// TIA Portal V17 export
// export: Created 2025-06-20T10:18:23.2551745Z, ExportSetting WithDefaults, DisplayName Totally Integrated Automation Portal, DisplayVersion V17 Update 8, DisplayName TIA Portal Openness, DisplayVersion V17 Update 8, DisplayName TIA Portal Version Control Interface, DisplayVersion V17, DisplayName SINAMICS Startdrive Advanced, DisplayVersion V17 SP2, DisplayName SINAMICS Startdrive G110M, G120, G120C, G120D, G120P, G115D, DisplayVersion V17 SP2, DisplayName SINAMICS Startdrive G130, G150, S120, S150, SINAMICS MV, S210, DisplayVersion V17 SP2, DisplayName STEP 7 Professional, DisplayVersion V17 Update 8, DisplayName SINUMERIK ONE STEP 7 Toolbox, DisplayVersion V17 Update 12, DisplayName SINUMERIK ONE PLC Basic Program Plus, DisplayVersion V17 Update 12, DisplayName SINUMERIK 840D sl STEP 7 Toolbox, DisplayVersion V17 Update 12, DisplayName STEP 7 Safety, DisplayVersion V17 Update 6, DisplayName WinCC Advanced, DisplayVersion V17 Update 8
FUNCTION "FC17000_MAIN_MAINTENANCE" : Void   // FC17000, LAD
{ S7_Optimized_Access := 'TRUE' }
VERSION : 0.1
// stored: AutoNumber false, IsIECCheckEnabled false, SetENOAutomatically false, UDAEnableTagReadback false
   VAR_TEMP
      ONLY_ONE_MAINT : Bool;
      NULL : Bool;
   END_VAR
BEGIN

REGION Network 1: CALL FC17100 MAINTENANCE HMI SCREEN VARIABLES
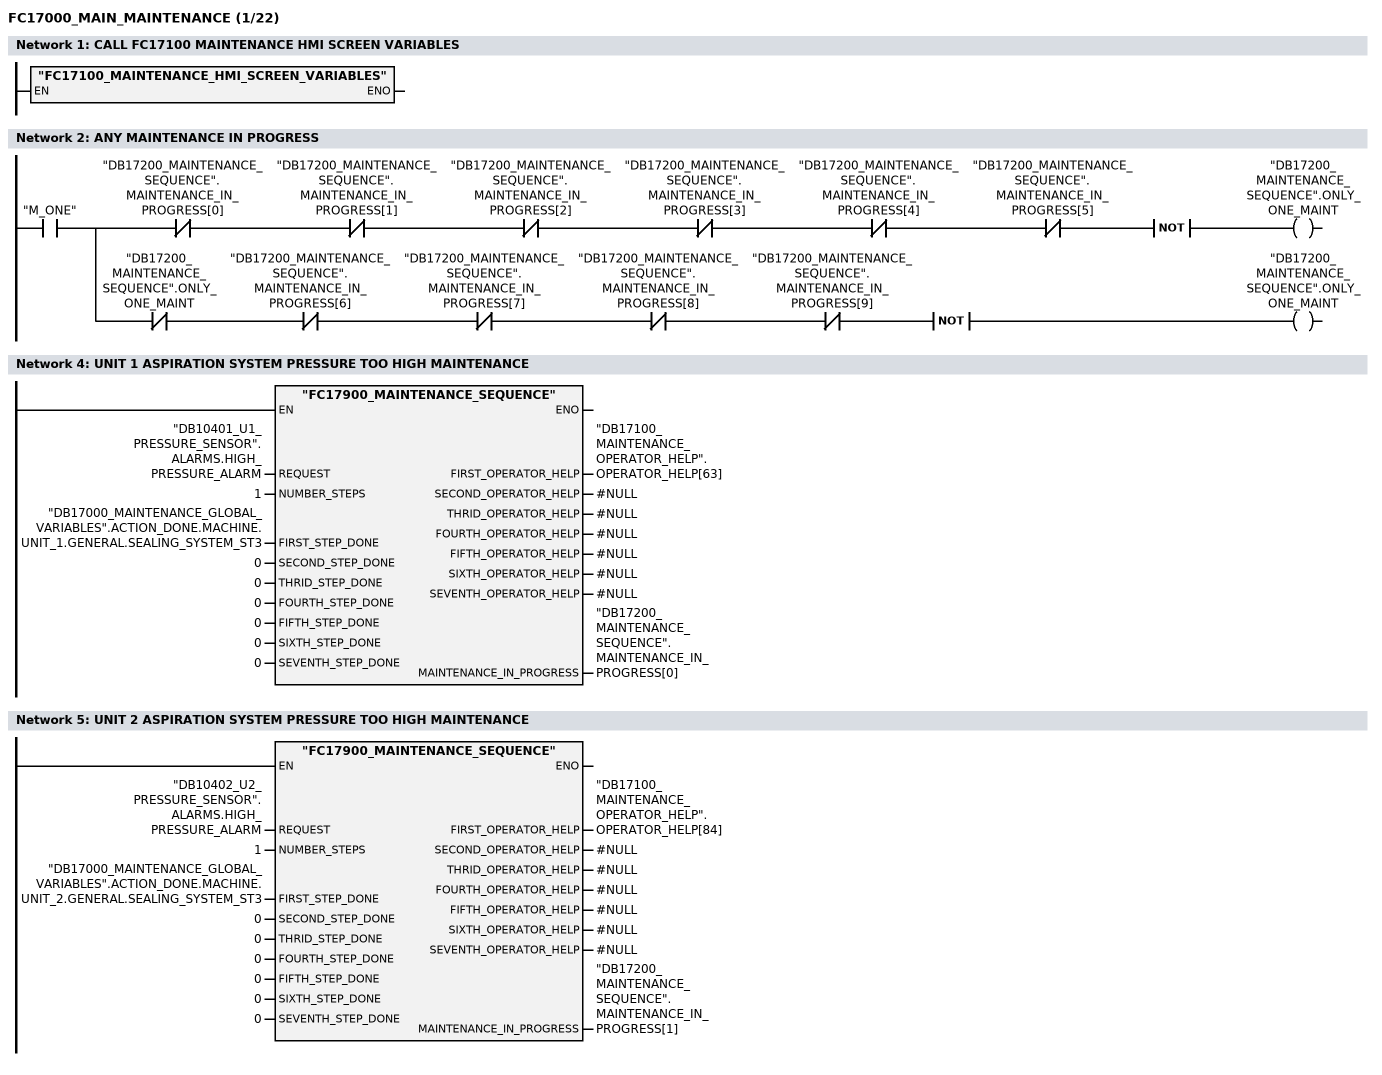
   RUNG wire#powerrail
      "FC17100_MAINTENANCE_HMI_SCREEN_VARIABLES"()
   END_RUNG
   // the same network as SCL:
   "FC17100_MAINTENANCE_HMI_SCREEN_VARIABLES"();
END_REGION

REGION Network 2: ANY MAINTENANCE IN PROGRESS
   RUNG wire#powerrail
      Contact( "M_ONE" )
      wire#w1
      I_Contact( "DB17200_MAINTENANCE_SEQUENCE".MAINTENANCE_IN_PROGRESS[0] )
      I_Contact( "DB17200_MAINTENANCE_SEQUENCE".MAINTENANCE_IN_PROGRESS[1] )
      I_Contact( "DB17200_MAINTENANCE_SEQUENCE".MAINTENANCE_IN_PROGRESS[2] )
      I_Contact( "DB17200_MAINTENANCE_SEQUENCE".MAINTENANCE_IN_PROGRESS[3] )
      I_Contact( "DB17200_MAINTENANCE_SEQUENCE".MAINTENANCE_IN_PROGRESS[4] )
      I_Contact( "DB17200_MAINTENANCE_SEQUENCE".MAINTENANCE_IN_PROGRESS[5] )
      Not()
      Coil( "DB17200_MAINTENANCE_SEQUENCE".ONLY_ONE_MAINT )
   END_RUNG
   RUNG wire#w1
      I_Contact( "DB17200_MAINTENANCE_SEQUENCE".ONLY_ONE_MAINT )
      I_Contact( "DB17200_MAINTENANCE_SEQUENCE".MAINTENANCE_IN_PROGRESS[6] )
      I_Contact( "DB17200_MAINTENANCE_SEQUENCE".MAINTENANCE_IN_PROGRESS[7] )
      I_Contact( "DB17200_MAINTENANCE_SEQUENCE".MAINTENANCE_IN_PROGRESS[8] )
      I_Contact( "DB17200_MAINTENANCE_SEQUENCE".MAINTENANCE_IN_PROGRESS[9] )
      Not()
      Coil( "DB17200_MAINTENANCE_SEQUENCE".ONLY_ONE_MAINT )
   END_RUNG
   // the same network as SCL:
   "DB17200_MAINTENANCE_SEQUENCE".ONLY_ONE_MAINT := NOT ("M_ONE" AND NOT "DB17200_MAINTENANCE_SEQUENCE".MAINTENANCE_IN_PROGRESS[0] AND NOT "DB17200_MAINTENANCE_SEQUENCE".MAINTENANCE_IN_PROGRESS[1] AND NOT "DB17200_MAINTENANCE_SEQUENCE".MAINTENANCE_IN_PROGRESS[2] AND NOT "DB17200_MAINTENANCE_SEQUENCE".MAINTENANCE_IN_PROGRESS[3] AND NOT "DB17200_MAINTENANCE_SEQUENCE".MAINTENANCE_IN_PROGRESS[4] AND NOT "DB17200_MAINTENANCE_SEQUENCE".MAINTENANCE_IN_PROGRESS[5]);
   "DB17200_MAINTENANCE_SEQUENCE".ONLY_ONE_MAINT := NOT ("M_ONE" AND NOT "DB17200_MAINTENANCE_SEQUENCE".ONLY_ONE_MAINT AND NOT "DB17200_MAINTENANCE_SEQUENCE".MAINTENANCE_IN_PROGRESS[6] AND NOT "DB17200_MAINTENANCE_SEQUENCE".MAINTENANCE_IN_PROGRESS[7] AND NOT "DB17200_MAINTENANCE_SEQUENCE".MAINTENANCE_IN_PROGRESS[8] AND NOT "DB17200_MAINTENANCE_SEQUENCE".MAINTENANCE_IN_PROGRESS[9]);
END_REGION

REGION Network 3: <<<---ALARMS--->>>
END_REGION

REGION Network 4: UNIT 1 ASPIRATION SYSTEM PRESSURE TOO HIGH MAINTENANCE
   RUNG wire#powerrail
      "FC17900_MAINTENANCE_SEQUENCE"(REQUEST := "DB10401_U1_PRESSURE_SENSOR".ALARMS.HIGH_PRESSURE_ALARM, NUMBER_STEPS := 1, FIRST_STEP_DONE := "DB17000_MAINTENANCE_GLOBAL_VARIABLES".ACTION_DONE.MACHINE.UNIT_1.GENERAL.SEALING_SYSTEM_ST3, SECOND_STEP_DONE := 0, THRID_STEP_DONE := 0, FOURTH_STEP_DONE := 0, FIFTH_STEP_DONE := 0, SIXTH_STEP_DONE := 0, SEVENTH_STEP_DONE := 0, FIRST_OPERATOR_HELP => "DB17100_MAINTENANCE_OPERATOR_HELP".OPERATOR_HELP[63], SECOND_OPERATOR_HELP => #NULL, THRID_OPERATOR_HELP => #NULL, FOURTH_OPERATOR_HELP => #NULL, FIFTH_OPERATOR_HELP => #NULL, SIXTH_OPERATOR_HELP => #NULL, SEVENTH_OPERATOR_HELP => #NULL, MAINTENANCE_IN_PROGRESS => "DB17200_MAINTENANCE_SEQUENCE".MAINTENANCE_IN_PROGRESS[0])
   END_RUNG
   // the same network as SCL:
   "FC17900_MAINTENANCE_SEQUENCE"(REQUEST := "DB10401_U1_PRESSURE_SENSOR".ALARMS.HIGH_PRESSURE_ALARM,
                           NUMBER_STEPS := 1,
                           FIRST_STEP_DONE := "DB17000_MAINTENANCE_GLOBAL_VARIABLES".ACTION_DONE.MACHINE.UNIT_1.GENERAL.SEALING_SYSTEM_ST3,
                           SECOND_STEP_DONE := 0,
                           THRID_STEP_DONE := 0,
                           FOURTH_STEP_DONE := 0,
                           FIFTH_STEP_DONE := 0,
                           SIXTH_STEP_DONE := 0,
                           SEVENTH_STEP_DONE := 0,
                           FIRST_OPERATOR_HELP => "DB17100_MAINTENANCE_OPERATOR_HELP".OPERATOR_HELP[63],
                           SECOND_OPERATOR_HELP => #NULL,
                           THRID_OPERATOR_HELP => #NULL,
                           FOURTH_OPERATOR_HELP => #NULL,
                           FIFTH_OPERATOR_HELP => #NULL,
                           SIXTH_OPERATOR_HELP => #NULL,
                           SEVENTH_OPERATOR_HELP => #NULL,
                           MAINTENANCE_IN_PROGRESS => "DB17200_MAINTENANCE_SEQUENCE".MAINTENANCE_IN_PROGRESS[0]);
END_REGION

REGION Network 5: UNIT 2 ASPIRATION SYSTEM PRESSURE TOO HIGH MAINTENANCE
   RUNG wire#powerrail
      "FC17900_MAINTENANCE_SEQUENCE"(REQUEST := "DB10402_U2_PRESSURE_SENSOR".ALARMS.HIGH_PRESSURE_ALARM, NUMBER_STEPS := 1, FIRST_STEP_DONE := "DB17000_MAINTENANCE_GLOBAL_VARIABLES".ACTION_DONE.MACHINE.UNIT_2.GENERAL.SEALING_SYSTEM_ST3, SECOND_STEP_DONE := 0, THRID_STEP_DONE := 0, FOURTH_STEP_DONE := 0, FIFTH_STEP_DONE := 0, SIXTH_STEP_DONE := 0, SEVENTH_STEP_DONE := 0, FIRST_OPERATOR_HELP => "DB17100_MAINTENANCE_OPERATOR_HELP".OPERATOR_HELP[84], SECOND_OPERATOR_HELP => #NULL, THRID_OPERATOR_HELP => #NULL, FOURTH_OPERATOR_HELP => #NULL, FIFTH_OPERATOR_HELP => #NULL, SIXTH_OPERATOR_HELP => #NULL, SEVENTH_OPERATOR_HELP => #NULL, MAINTENANCE_IN_PROGRESS => "DB17200_MAINTENANCE_SEQUENCE".MAINTENANCE_IN_PROGRESS[1])
   END_RUNG
   // the same network as SCL:
   "FC17900_MAINTENANCE_SEQUENCE"(REQUEST := "DB10402_U2_PRESSURE_SENSOR".ALARMS.HIGH_PRESSURE_ALARM,
                           NUMBER_STEPS := 1,
                           FIRST_STEP_DONE := "DB17000_MAINTENANCE_GLOBAL_VARIABLES".ACTION_DONE.MACHINE.UNIT_2.GENERAL.SEALING_SYSTEM_ST3,
                           SECOND_STEP_DONE := 0,
                           THRID_STEP_DONE := 0,
                           FOURTH_STEP_DONE := 0,
                           FIFTH_STEP_DONE := 0,
                           SIXTH_STEP_DONE := 0,
                           SEVENTH_STEP_DONE := 0,
                           FIRST_OPERATOR_HELP => "DB17100_MAINTENANCE_OPERATOR_HELP".OPERATOR_HELP[84],
                           SECOND_OPERATOR_HELP => #NULL,
                           THRID_OPERATOR_HELP => #NULL,
                           FOURTH_OPERATOR_HELP => #NULL,
                           FIFTH_OPERATOR_HELP => #NULL,
                           SIXTH_OPERATOR_HELP => #NULL,
                           SEVENTH_OPERATOR_HELP => #NULL,
                           MAINTENANCE_IN_PROGRESS => "DB17200_MAINTENANCE_SEQUENCE".MAINTENANCE_IN_PROGRESS[1]);
END_REGION

REGION Network 6: UNIT 1 FIXTURE 1 NOT CLAMPED
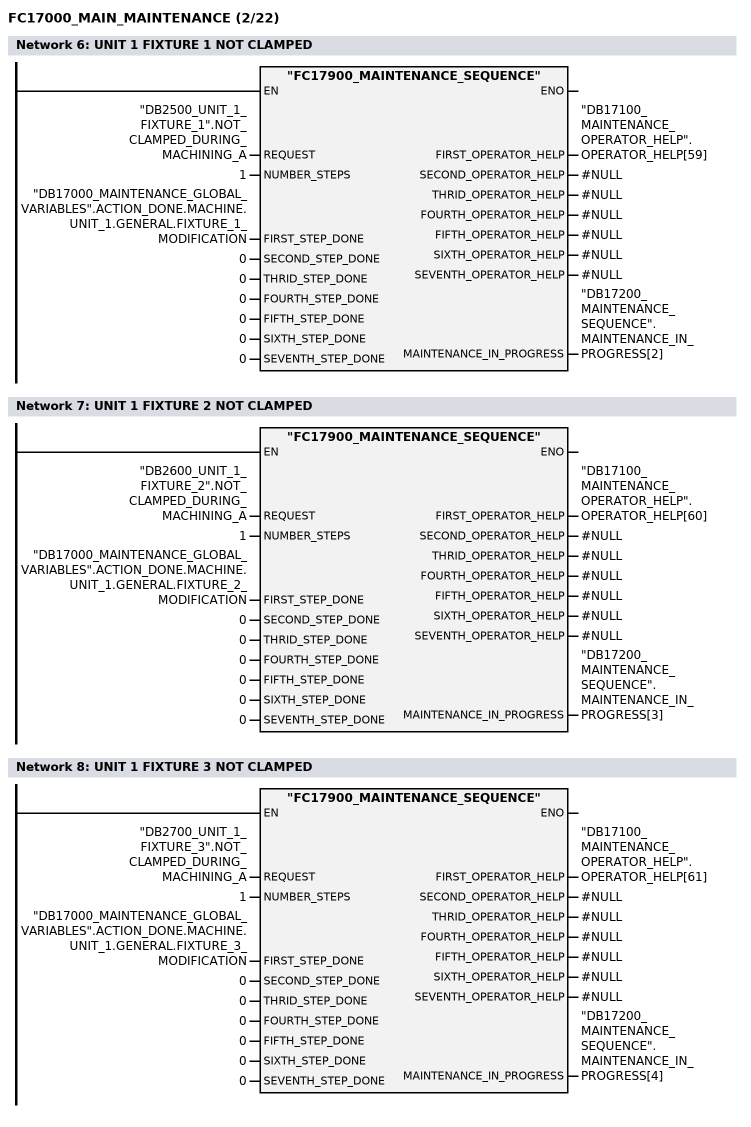
   RUNG wire#powerrail
      "FC17900_MAINTENANCE_SEQUENCE"(REQUEST := "DB2500_UNIT_1_FIXTURE_1".NOT_CLAMPED_DURING_MACHINING_A, NUMBER_STEPS := 1, FIRST_STEP_DONE := "DB17000_MAINTENANCE_GLOBAL_VARIABLES".ACTION_DONE.MACHINE.UNIT_1.GENERAL.FIXTURE_1_MODIFICATION, SECOND_STEP_DONE := 0, THRID_STEP_DONE := 0, FOURTH_STEP_DONE := 0, FIFTH_STEP_DONE := 0, SIXTH_STEP_DONE := 0, SEVENTH_STEP_DONE := 0, FIRST_OPERATOR_HELP => "DB17100_MAINTENANCE_OPERATOR_HELP".OPERATOR_HELP[59], SECOND_OPERATOR_HELP => #NULL, THRID_OPERATOR_HELP => #NULL, FOURTH_OPERATOR_HELP => #NULL, FIFTH_OPERATOR_HELP => #NULL, SIXTH_OPERATOR_HELP => #NULL, SEVENTH_OPERATOR_HELP => #NULL, MAINTENANCE_IN_PROGRESS => "DB17200_MAINTENANCE_SEQUENCE".MAINTENANCE_IN_PROGRESS[2])
   END_RUNG
   // the same network as SCL:
   "FC17900_MAINTENANCE_SEQUENCE"(REQUEST := "DB2500_UNIT_1_FIXTURE_1".NOT_CLAMPED_DURING_MACHINING_A,
                           NUMBER_STEPS := 1,
                           FIRST_STEP_DONE := "DB17000_MAINTENANCE_GLOBAL_VARIABLES".ACTION_DONE.MACHINE.UNIT_1.GENERAL.FIXTURE_1_MODIFICATION,
                           SECOND_STEP_DONE := 0,
                           THRID_STEP_DONE := 0,
                           FOURTH_STEP_DONE := 0,
                           FIFTH_STEP_DONE := 0,
                           SIXTH_STEP_DONE := 0,
                           SEVENTH_STEP_DONE := 0,
                           FIRST_OPERATOR_HELP => "DB17100_MAINTENANCE_OPERATOR_HELP".OPERATOR_HELP[59],
                           SECOND_OPERATOR_HELP => #NULL,
                           THRID_OPERATOR_HELP => #NULL,
                           FOURTH_OPERATOR_HELP => #NULL,
                           FIFTH_OPERATOR_HELP => #NULL,
                           SIXTH_OPERATOR_HELP => #NULL,
                           SEVENTH_OPERATOR_HELP => #NULL,
                           MAINTENANCE_IN_PROGRESS => "DB17200_MAINTENANCE_SEQUENCE".MAINTENANCE_IN_PROGRESS[2]);
END_REGION

REGION Network 7: UNIT 1 FIXTURE 2 NOT CLAMPED
   RUNG wire#powerrail
      "FC17900_MAINTENANCE_SEQUENCE"(REQUEST := "DB2600_UNIT_1_FIXTURE_2".NOT_CLAMPED_DURING_MACHINING_A, NUMBER_STEPS := 1, FIRST_STEP_DONE := "DB17000_MAINTENANCE_GLOBAL_VARIABLES".ACTION_DONE.MACHINE.UNIT_1.GENERAL.FIXTURE_2_MODIFICATION, SECOND_STEP_DONE := 0, THRID_STEP_DONE := 0, FOURTH_STEP_DONE := 0, FIFTH_STEP_DONE := 0, SIXTH_STEP_DONE := 0, SEVENTH_STEP_DONE := 0, FIRST_OPERATOR_HELP => "DB17100_MAINTENANCE_OPERATOR_HELP".OPERATOR_HELP[60], SECOND_OPERATOR_HELP => #NULL, THRID_OPERATOR_HELP => #NULL, FOURTH_OPERATOR_HELP => #NULL, FIFTH_OPERATOR_HELP => #NULL, SIXTH_OPERATOR_HELP => #NULL, SEVENTH_OPERATOR_HELP => #NULL, MAINTENANCE_IN_PROGRESS => "DB17200_MAINTENANCE_SEQUENCE".MAINTENANCE_IN_PROGRESS[3])
   END_RUNG
   // the same network as SCL:
   "FC17900_MAINTENANCE_SEQUENCE"(REQUEST := "DB2600_UNIT_1_FIXTURE_2".NOT_CLAMPED_DURING_MACHINING_A,
                           NUMBER_STEPS := 1,
                           FIRST_STEP_DONE := "DB17000_MAINTENANCE_GLOBAL_VARIABLES".ACTION_DONE.MACHINE.UNIT_1.GENERAL.FIXTURE_2_MODIFICATION,
                           SECOND_STEP_DONE := 0,
                           THRID_STEP_DONE := 0,
                           FOURTH_STEP_DONE := 0,
                           FIFTH_STEP_DONE := 0,
                           SIXTH_STEP_DONE := 0,
                           SEVENTH_STEP_DONE := 0,
                           FIRST_OPERATOR_HELP => "DB17100_MAINTENANCE_OPERATOR_HELP".OPERATOR_HELP[60],
                           SECOND_OPERATOR_HELP => #NULL,
                           THRID_OPERATOR_HELP => #NULL,
                           FOURTH_OPERATOR_HELP => #NULL,
                           FIFTH_OPERATOR_HELP => #NULL,
                           SIXTH_OPERATOR_HELP => #NULL,
                           SEVENTH_OPERATOR_HELP => #NULL,
                           MAINTENANCE_IN_PROGRESS => "DB17200_MAINTENANCE_SEQUENCE".MAINTENANCE_IN_PROGRESS[3]);
END_REGION

REGION Network 8: UNIT 1 FIXTURE 3 NOT CLAMPED
   RUNG wire#powerrail
      "FC17900_MAINTENANCE_SEQUENCE"(REQUEST := "DB2700_UNIT_1_FIXTURE_3".NOT_CLAMPED_DURING_MACHINING_A, NUMBER_STEPS := 1, FIRST_STEP_DONE := "DB17000_MAINTENANCE_GLOBAL_VARIABLES".ACTION_DONE.MACHINE.UNIT_1.GENERAL.FIXTURE_3_MODIFICATION, SECOND_STEP_DONE := 0, THRID_STEP_DONE := 0, FOURTH_STEP_DONE := 0, FIFTH_STEP_DONE := 0, SIXTH_STEP_DONE := 0, SEVENTH_STEP_DONE := 0, FIRST_OPERATOR_HELP => "DB17100_MAINTENANCE_OPERATOR_HELP".OPERATOR_HELP[61], SECOND_OPERATOR_HELP => #NULL, THRID_OPERATOR_HELP => #NULL, FOURTH_OPERATOR_HELP => #NULL, FIFTH_OPERATOR_HELP => #NULL, SIXTH_OPERATOR_HELP => #NULL, SEVENTH_OPERATOR_HELP => #NULL, MAINTENANCE_IN_PROGRESS => "DB17200_MAINTENANCE_SEQUENCE".MAINTENANCE_IN_PROGRESS[4])
   END_RUNG
   // the same network as SCL:
   "FC17900_MAINTENANCE_SEQUENCE"(REQUEST := "DB2700_UNIT_1_FIXTURE_3".NOT_CLAMPED_DURING_MACHINING_A,
                           NUMBER_STEPS := 1,
                           FIRST_STEP_DONE := "DB17000_MAINTENANCE_GLOBAL_VARIABLES".ACTION_DONE.MACHINE.UNIT_1.GENERAL.FIXTURE_3_MODIFICATION,
                           SECOND_STEP_DONE := 0,
                           THRID_STEP_DONE := 0,
                           FOURTH_STEP_DONE := 0,
                           FIFTH_STEP_DONE := 0,
                           SIXTH_STEP_DONE := 0,
                           SEVENTH_STEP_DONE := 0,
                           FIRST_OPERATOR_HELP => "DB17100_MAINTENANCE_OPERATOR_HELP".OPERATOR_HELP[61],
                           SECOND_OPERATOR_HELP => #NULL,
                           THRID_OPERATOR_HELP => #NULL,
                           FOURTH_OPERATOR_HELP => #NULL,
                           FIFTH_OPERATOR_HELP => #NULL,
                           SIXTH_OPERATOR_HELP => #NULL,
                           SEVENTH_OPERATOR_HELP => #NULL,
                           MAINTENANCE_IN_PROGRESS => "DB17200_MAINTENANCE_SEQUENCE".MAINTENANCE_IN_PROGRESS[4]);
END_REGION

REGION Network 9: UNIT 1 FIXTURE 4 NOT CLAMPED
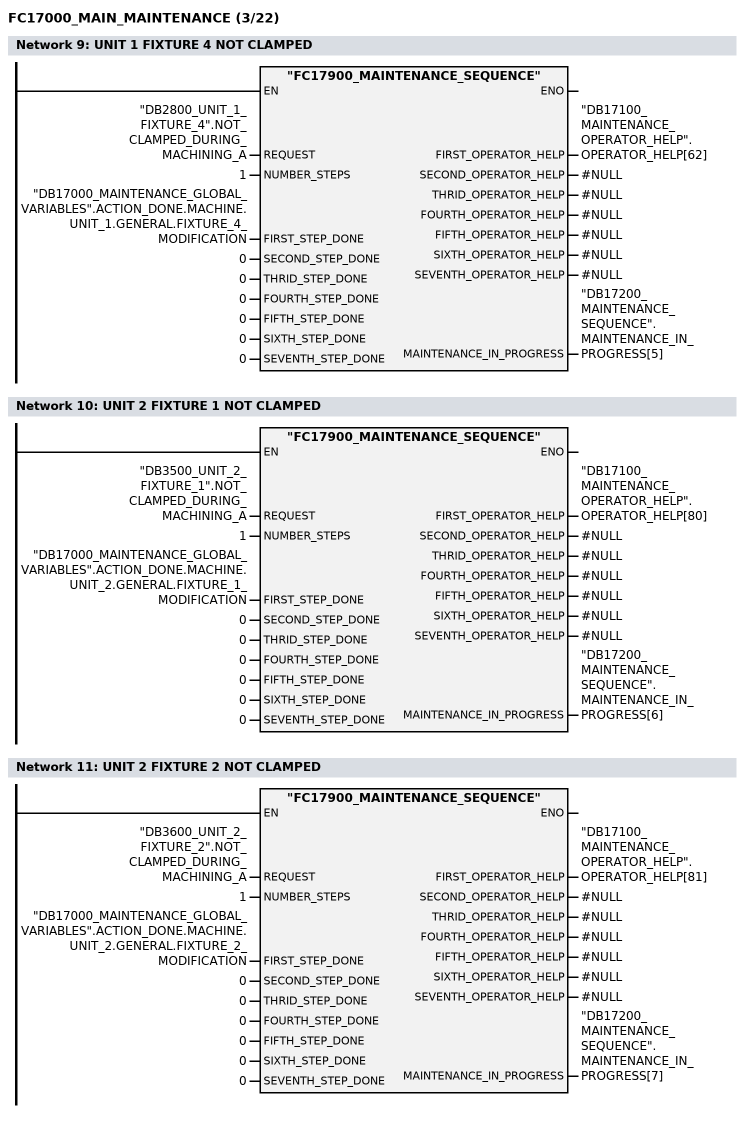
   RUNG wire#powerrail
      "FC17900_MAINTENANCE_SEQUENCE"(REQUEST := "DB2800_UNIT_1_FIXTURE_4".NOT_CLAMPED_DURING_MACHINING_A, NUMBER_STEPS := 1, FIRST_STEP_DONE := "DB17000_MAINTENANCE_GLOBAL_VARIABLES".ACTION_DONE.MACHINE.UNIT_1.GENERAL.FIXTURE_4_MODIFICATION, SECOND_STEP_DONE := 0, THRID_STEP_DONE := 0, FOURTH_STEP_DONE := 0, FIFTH_STEP_DONE := 0, SIXTH_STEP_DONE := 0, SEVENTH_STEP_DONE := 0, FIRST_OPERATOR_HELP => "DB17100_MAINTENANCE_OPERATOR_HELP".OPERATOR_HELP[62], SECOND_OPERATOR_HELP => #NULL, THRID_OPERATOR_HELP => #NULL, FOURTH_OPERATOR_HELP => #NULL, FIFTH_OPERATOR_HELP => #NULL, SIXTH_OPERATOR_HELP => #NULL, SEVENTH_OPERATOR_HELP => #NULL, MAINTENANCE_IN_PROGRESS => "DB17200_MAINTENANCE_SEQUENCE".MAINTENANCE_IN_PROGRESS[5])
   END_RUNG
   // the same network as SCL:
   "FC17900_MAINTENANCE_SEQUENCE"(REQUEST := "DB2800_UNIT_1_FIXTURE_4".NOT_CLAMPED_DURING_MACHINING_A,
                           NUMBER_STEPS := 1,
                           FIRST_STEP_DONE := "DB17000_MAINTENANCE_GLOBAL_VARIABLES".ACTION_DONE.MACHINE.UNIT_1.GENERAL.FIXTURE_4_MODIFICATION,
                           SECOND_STEP_DONE := 0,
                           THRID_STEP_DONE := 0,
                           FOURTH_STEP_DONE := 0,
                           FIFTH_STEP_DONE := 0,
                           SIXTH_STEP_DONE := 0,
                           SEVENTH_STEP_DONE := 0,
                           FIRST_OPERATOR_HELP => "DB17100_MAINTENANCE_OPERATOR_HELP".OPERATOR_HELP[62],
                           SECOND_OPERATOR_HELP => #NULL,
                           THRID_OPERATOR_HELP => #NULL,
                           FOURTH_OPERATOR_HELP => #NULL,
                           FIFTH_OPERATOR_HELP => #NULL,
                           SIXTH_OPERATOR_HELP => #NULL,
                           SEVENTH_OPERATOR_HELP => #NULL,
                           MAINTENANCE_IN_PROGRESS => "DB17200_MAINTENANCE_SEQUENCE".MAINTENANCE_IN_PROGRESS[5]);
END_REGION

REGION Network 10: UNIT 2 FIXTURE 1 NOT CLAMPED
   RUNG wire#powerrail
      "FC17900_MAINTENANCE_SEQUENCE"(REQUEST := "DB3500_UNIT_2_FIXTURE_1".NOT_CLAMPED_DURING_MACHINING_A, NUMBER_STEPS := 1, FIRST_STEP_DONE := "DB17000_MAINTENANCE_GLOBAL_VARIABLES".ACTION_DONE.MACHINE.UNIT_2.GENERAL.FIXTURE_1_MODIFICATION, SECOND_STEP_DONE := 0, THRID_STEP_DONE := 0, FOURTH_STEP_DONE := 0, FIFTH_STEP_DONE := 0, SIXTH_STEP_DONE := 0, SEVENTH_STEP_DONE := 0, FIRST_OPERATOR_HELP => "DB17100_MAINTENANCE_OPERATOR_HELP".OPERATOR_HELP[80], SECOND_OPERATOR_HELP => #NULL, THRID_OPERATOR_HELP => #NULL, FOURTH_OPERATOR_HELP => #NULL, FIFTH_OPERATOR_HELP => #NULL, SIXTH_OPERATOR_HELP => #NULL, SEVENTH_OPERATOR_HELP => #NULL, MAINTENANCE_IN_PROGRESS => "DB17200_MAINTENANCE_SEQUENCE".MAINTENANCE_IN_PROGRESS[6])
   END_RUNG
   // the same network as SCL:
   "FC17900_MAINTENANCE_SEQUENCE"(REQUEST := "DB3500_UNIT_2_FIXTURE_1".NOT_CLAMPED_DURING_MACHINING_A,
                           NUMBER_STEPS := 1,
                           FIRST_STEP_DONE := "DB17000_MAINTENANCE_GLOBAL_VARIABLES".ACTION_DONE.MACHINE.UNIT_2.GENERAL.FIXTURE_1_MODIFICATION,
                           SECOND_STEP_DONE := 0,
                           THRID_STEP_DONE := 0,
                           FOURTH_STEP_DONE := 0,
                           FIFTH_STEP_DONE := 0,
                           SIXTH_STEP_DONE := 0,
                           SEVENTH_STEP_DONE := 0,
                           FIRST_OPERATOR_HELP => "DB17100_MAINTENANCE_OPERATOR_HELP".OPERATOR_HELP[80],
                           SECOND_OPERATOR_HELP => #NULL,
                           THRID_OPERATOR_HELP => #NULL,
                           FOURTH_OPERATOR_HELP => #NULL,
                           FIFTH_OPERATOR_HELP => #NULL,
                           SIXTH_OPERATOR_HELP => #NULL,
                           SEVENTH_OPERATOR_HELP => #NULL,
                           MAINTENANCE_IN_PROGRESS => "DB17200_MAINTENANCE_SEQUENCE".MAINTENANCE_IN_PROGRESS[6]);
END_REGION

REGION Network 11: UNIT 2 FIXTURE 2 NOT CLAMPED
   RUNG wire#powerrail
      "FC17900_MAINTENANCE_SEQUENCE"(REQUEST := "DB3600_UNIT_2_FIXTURE_2".NOT_CLAMPED_DURING_MACHINING_A, NUMBER_STEPS := 1, FIRST_STEP_DONE := "DB17000_MAINTENANCE_GLOBAL_VARIABLES".ACTION_DONE.MACHINE.UNIT_2.GENERAL.FIXTURE_2_MODIFICATION, SECOND_STEP_DONE := 0, THRID_STEP_DONE := 0, FOURTH_STEP_DONE := 0, FIFTH_STEP_DONE := 0, SIXTH_STEP_DONE := 0, SEVENTH_STEP_DONE := 0, FIRST_OPERATOR_HELP => "DB17100_MAINTENANCE_OPERATOR_HELP".OPERATOR_HELP[81], SECOND_OPERATOR_HELP => #NULL, THRID_OPERATOR_HELP => #NULL, FOURTH_OPERATOR_HELP => #NULL, FIFTH_OPERATOR_HELP => #NULL, SIXTH_OPERATOR_HELP => #NULL, SEVENTH_OPERATOR_HELP => #NULL, MAINTENANCE_IN_PROGRESS => "DB17200_MAINTENANCE_SEQUENCE".MAINTENANCE_IN_PROGRESS[7])
   END_RUNG
   // the same network as SCL:
   "FC17900_MAINTENANCE_SEQUENCE"(REQUEST := "DB3600_UNIT_2_FIXTURE_2".NOT_CLAMPED_DURING_MACHINING_A,
                           NUMBER_STEPS := 1,
                           FIRST_STEP_DONE := "DB17000_MAINTENANCE_GLOBAL_VARIABLES".ACTION_DONE.MACHINE.UNIT_2.GENERAL.FIXTURE_2_MODIFICATION,
                           SECOND_STEP_DONE := 0,
                           THRID_STEP_DONE := 0,
                           FOURTH_STEP_DONE := 0,
                           FIFTH_STEP_DONE := 0,
                           SIXTH_STEP_DONE := 0,
                           SEVENTH_STEP_DONE := 0,
                           FIRST_OPERATOR_HELP => "DB17100_MAINTENANCE_OPERATOR_HELP".OPERATOR_HELP[81],
                           SECOND_OPERATOR_HELP => #NULL,
                           THRID_OPERATOR_HELP => #NULL,
                           FOURTH_OPERATOR_HELP => #NULL,
                           FIFTH_OPERATOR_HELP => #NULL,
                           SIXTH_OPERATOR_HELP => #NULL,
                           SEVENTH_OPERATOR_HELP => #NULL,
                           MAINTENANCE_IN_PROGRESS => "DB17200_MAINTENANCE_SEQUENCE".MAINTENANCE_IN_PROGRESS[7]);
END_REGION

REGION Network 12: UNIT 2 FIXTURE 3 NOT CLAMPED
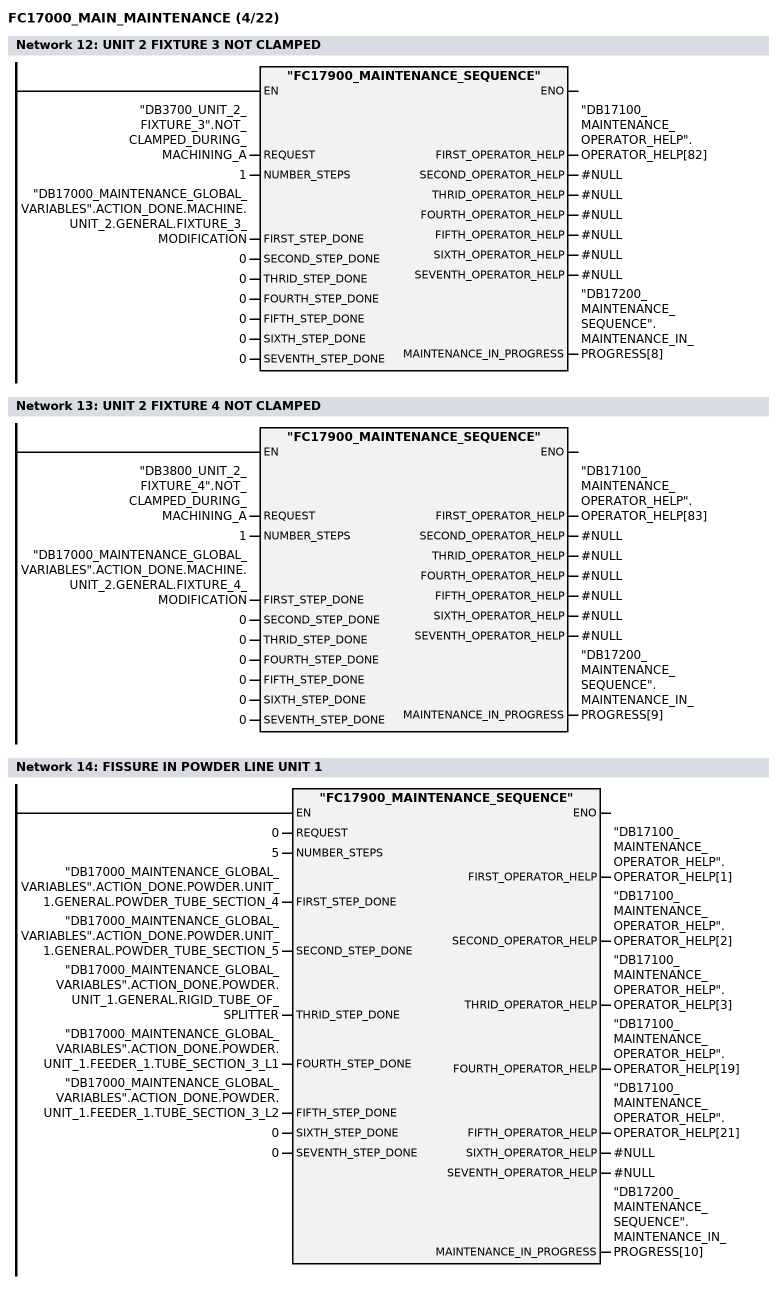
   RUNG wire#powerrail
      "FC17900_MAINTENANCE_SEQUENCE"(REQUEST := "DB3700_UNIT_2_FIXTURE_3".NOT_CLAMPED_DURING_MACHINING_A, NUMBER_STEPS := 1, FIRST_STEP_DONE := "DB17000_MAINTENANCE_GLOBAL_VARIABLES".ACTION_DONE.MACHINE.UNIT_2.GENERAL.FIXTURE_3_MODIFICATION, SECOND_STEP_DONE := 0, THRID_STEP_DONE := 0, FOURTH_STEP_DONE := 0, FIFTH_STEP_DONE := 0, SIXTH_STEP_DONE := 0, SEVENTH_STEP_DONE := 0, FIRST_OPERATOR_HELP => "DB17100_MAINTENANCE_OPERATOR_HELP".OPERATOR_HELP[82], SECOND_OPERATOR_HELP => #NULL, THRID_OPERATOR_HELP => #NULL, FOURTH_OPERATOR_HELP => #NULL, FIFTH_OPERATOR_HELP => #NULL, SIXTH_OPERATOR_HELP => #NULL, SEVENTH_OPERATOR_HELP => #NULL, MAINTENANCE_IN_PROGRESS => "DB17200_MAINTENANCE_SEQUENCE".MAINTENANCE_IN_PROGRESS[8])
   END_RUNG
   // the same network as SCL:
   "FC17900_MAINTENANCE_SEQUENCE"(REQUEST := "DB3700_UNIT_2_FIXTURE_3".NOT_CLAMPED_DURING_MACHINING_A,
                           NUMBER_STEPS := 1,
                           FIRST_STEP_DONE := "DB17000_MAINTENANCE_GLOBAL_VARIABLES".ACTION_DONE.MACHINE.UNIT_2.GENERAL.FIXTURE_3_MODIFICATION,
                           SECOND_STEP_DONE := 0,
                           THRID_STEP_DONE := 0,
                           FOURTH_STEP_DONE := 0,
                           FIFTH_STEP_DONE := 0,
                           SIXTH_STEP_DONE := 0,
                           SEVENTH_STEP_DONE := 0,
                           FIRST_OPERATOR_HELP => "DB17100_MAINTENANCE_OPERATOR_HELP".OPERATOR_HELP[82],
                           SECOND_OPERATOR_HELP => #NULL,
                           THRID_OPERATOR_HELP => #NULL,
                           FOURTH_OPERATOR_HELP => #NULL,
                           FIFTH_OPERATOR_HELP => #NULL,
                           SIXTH_OPERATOR_HELP => #NULL,
                           SEVENTH_OPERATOR_HELP => #NULL,
                           MAINTENANCE_IN_PROGRESS => "DB17200_MAINTENANCE_SEQUENCE".MAINTENANCE_IN_PROGRESS[8]);
END_REGION

REGION Network 13: UNIT 2 FIXTURE 4 NOT CLAMPED
   RUNG wire#powerrail
      "FC17900_MAINTENANCE_SEQUENCE"(REQUEST := "DB3800_UNIT_2_FIXTURE_4".NOT_CLAMPED_DURING_MACHINING_A, NUMBER_STEPS := 1, FIRST_STEP_DONE := "DB17000_MAINTENANCE_GLOBAL_VARIABLES".ACTION_DONE.MACHINE.UNIT_2.GENERAL.FIXTURE_4_MODIFICATION, SECOND_STEP_DONE := 0, THRID_STEP_DONE := 0, FOURTH_STEP_DONE := 0, FIFTH_STEP_DONE := 0, SIXTH_STEP_DONE := 0, SEVENTH_STEP_DONE := 0, FIRST_OPERATOR_HELP => "DB17100_MAINTENANCE_OPERATOR_HELP".OPERATOR_HELP[83], SECOND_OPERATOR_HELP => #NULL, THRID_OPERATOR_HELP => #NULL, FOURTH_OPERATOR_HELP => #NULL, FIFTH_OPERATOR_HELP => #NULL, SIXTH_OPERATOR_HELP => #NULL, SEVENTH_OPERATOR_HELP => #NULL, MAINTENANCE_IN_PROGRESS => "DB17200_MAINTENANCE_SEQUENCE".MAINTENANCE_IN_PROGRESS[9])
   END_RUNG
   // the same network as SCL:
   "FC17900_MAINTENANCE_SEQUENCE"(REQUEST := "DB3800_UNIT_2_FIXTURE_4".NOT_CLAMPED_DURING_MACHINING_A,
                           NUMBER_STEPS := 1,
                           FIRST_STEP_DONE := "DB17000_MAINTENANCE_GLOBAL_VARIABLES".ACTION_DONE.MACHINE.UNIT_2.GENERAL.FIXTURE_4_MODIFICATION,
                           SECOND_STEP_DONE := 0,
                           THRID_STEP_DONE := 0,
                           FOURTH_STEP_DONE := 0,
                           FIFTH_STEP_DONE := 0,
                           SIXTH_STEP_DONE := 0,
                           SEVENTH_STEP_DONE := 0,
                           FIRST_OPERATOR_HELP => "DB17100_MAINTENANCE_OPERATOR_HELP".OPERATOR_HELP[83],
                           SECOND_OPERATOR_HELP => #NULL,
                           THRID_OPERATOR_HELP => #NULL,
                           FOURTH_OPERATOR_HELP => #NULL,
                           FIFTH_OPERATOR_HELP => #NULL,
                           SIXTH_OPERATOR_HELP => #NULL,
                           SEVENTH_OPERATOR_HELP => #NULL,
                           MAINTENANCE_IN_PROGRESS => "DB17200_MAINTENANCE_SEQUENCE".MAINTENANCE_IN_PROGRESS[9]);
END_REGION

REGION Network 14: FISSURE IN POWDER LINE UNIT 1
   RUNG wire#powerrail
      "FC17900_MAINTENANCE_SEQUENCE"(REQUEST := 0, NUMBER_STEPS := 5, FIRST_STEP_DONE := "DB17000_MAINTENANCE_GLOBAL_VARIABLES".ACTION_DONE.POWDER.UNIT_1.GENERAL.POWDER_TUBE_SECTION_4, SECOND_STEP_DONE := "DB17000_MAINTENANCE_GLOBAL_VARIABLES".ACTION_DONE.POWDER.UNIT_1.GENERAL.POWDER_TUBE_SECTION_5, THRID_STEP_DONE := "DB17000_MAINTENANCE_GLOBAL_VARIABLES".ACTION_DONE.POWDER.UNIT_1.GENERAL.RIGID_TUBE_OF_SPLITTER, FOURTH_STEP_DONE := "DB17000_MAINTENANCE_GLOBAL_VARIABLES".ACTION_DONE.POWDER.UNIT_1.FEEDER_1.TUBE_SECTION_3_L1, FIFTH_STEP_DONE := "DB17000_MAINTENANCE_GLOBAL_VARIABLES".ACTION_DONE.POWDER.UNIT_1.FEEDER_1.TUBE_SECTION_3_L2, SIXTH_STEP_DONE := 0, SEVENTH_STEP_DONE := 0, FIRST_OPERATOR_HELP => "DB17100_MAINTENANCE_OPERATOR_HELP".OPERATOR_HELP[1], SECOND_OPERATOR_HELP => "DB17100_MAINTENANCE_OPERATOR_HELP".OPERATOR_HELP[2], THRID_OPERATOR_HELP => "DB17100_MAINTENANCE_OPERATOR_HELP".OPERATOR_HELP[3], FOURTH_OPERATOR_HELP => "DB17100_MAINTENANCE_OPERATOR_HELP".OPERATOR_HELP[19], FIFTH_OPERATOR_HELP => "DB17100_MAINTENANCE_OPERATOR_HELP".OPERATOR_HELP[21], SIXTH_OPERATOR_HELP => #NULL, SEVENTH_OPERATOR_HELP => #NULL, MAINTENANCE_IN_PROGRESS => "DB17200_MAINTENANCE_SEQUENCE".MAINTENANCE_IN_PROGRESS[10])
   END_RUNG
   // the same network as SCL:
   "FC17900_MAINTENANCE_SEQUENCE"(REQUEST := 0,
                           NUMBER_STEPS := 5,
                           FIRST_STEP_DONE := "DB17000_MAINTENANCE_GLOBAL_VARIABLES".ACTION_DONE.POWDER.UNIT_1.GENERAL.POWDER_TUBE_SECTION_4,
                           SECOND_STEP_DONE := "DB17000_MAINTENANCE_GLOBAL_VARIABLES".ACTION_DONE.POWDER.UNIT_1.GENERAL.POWDER_TUBE_SECTION_5,
                           THRID_STEP_DONE := "DB17000_MAINTENANCE_GLOBAL_VARIABLES".ACTION_DONE.POWDER.UNIT_1.GENERAL.RIGID_TUBE_OF_SPLITTER,
                           FOURTH_STEP_DONE := "DB17000_MAINTENANCE_GLOBAL_VARIABLES".ACTION_DONE.POWDER.UNIT_1.FEEDER_1.TUBE_SECTION_3_L1,
                           FIFTH_STEP_DONE := "DB17000_MAINTENANCE_GLOBAL_VARIABLES".ACTION_DONE.POWDER.UNIT_1.FEEDER_1.TUBE_SECTION_3_L2,
                           SIXTH_STEP_DONE := 0,
                           SEVENTH_STEP_DONE := 0,
                           FIRST_OPERATOR_HELP => "DB17100_MAINTENANCE_OPERATOR_HELP".OPERATOR_HELP[1],
                           SECOND_OPERATOR_HELP => "DB17100_MAINTENANCE_OPERATOR_HELP".OPERATOR_HELP[2],
                           THRID_OPERATOR_HELP => "DB17100_MAINTENANCE_OPERATOR_HELP".OPERATOR_HELP[3],
                           FOURTH_OPERATOR_HELP => "DB17100_MAINTENANCE_OPERATOR_HELP".OPERATOR_HELP[19],
                           FIFTH_OPERATOR_HELP => "DB17100_MAINTENANCE_OPERATOR_HELP".OPERATOR_HELP[21],
                           SIXTH_OPERATOR_HELP => #NULL,
                           SEVENTH_OPERATOR_HELP => #NULL,
                           MAINTENANCE_IN_PROGRESS => "DB17200_MAINTENANCE_SEQUENCE".MAINTENANCE_IN_PROGRESS[10]);
END_REGION

REGION Network 15: FISSURE IN POWDER LINE UNIT 2
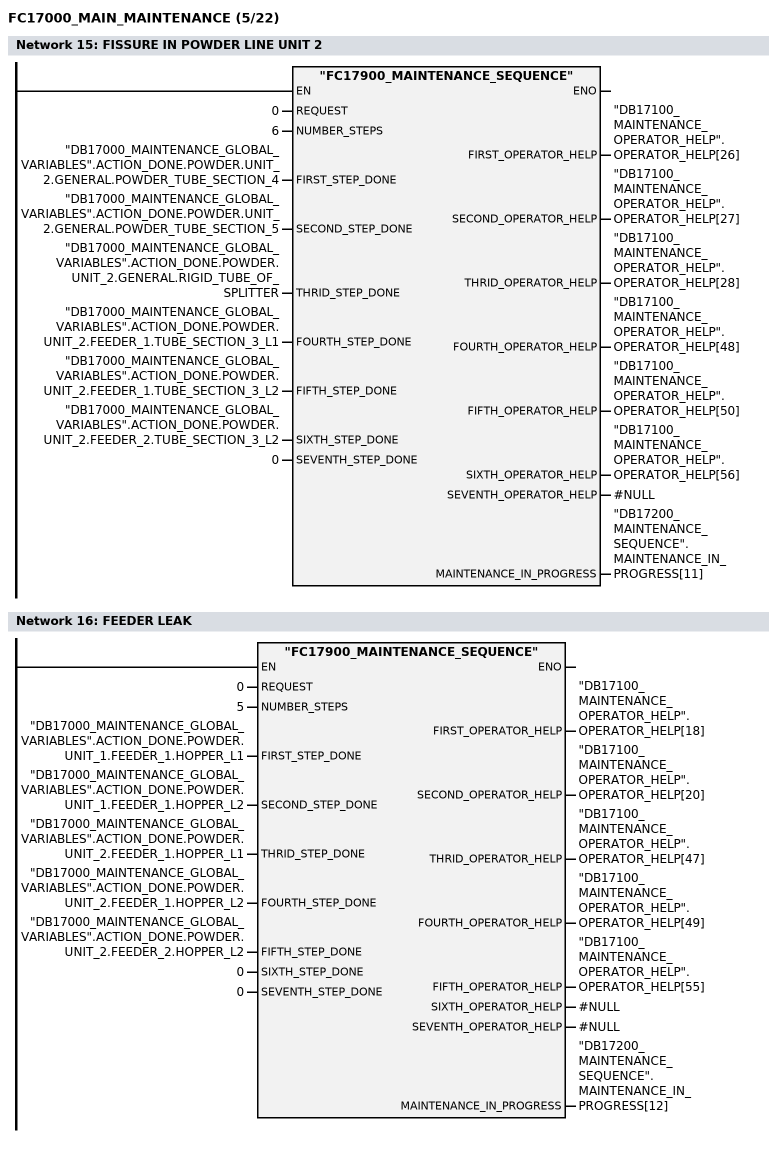
   RUNG wire#powerrail
      "FC17900_MAINTENANCE_SEQUENCE"(REQUEST := 0, NUMBER_STEPS := 6, FIRST_STEP_DONE := "DB17000_MAINTENANCE_GLOBAL_VARIABLES".ACTION_DONE.POWDER.UNIT_2.GENERAL.POWDER_TUBE_SECTION_4, SECOND_STEP_DONE := "DB17000_MAINTENANCE_GLOBAL_VARIABLES".ACTION_DONE.POWDER.UNIT_2.GENERAL.POWDER_TUBE_SECTION_5, THRID_STEP_DONE := "DB17000_MAINTENANCE_GLOBAL_VARIABLES".ACTION_DONE.POWDER.UNIT_2.GENERAL.RIGID_TUBE_OF_SPLITTER, FOURTH_STEP_DONE := "DB17000_MAINTENANCE_GLOBAL_VARIABLES".ACTION_DONE.POWDER.UNIT_2.FEEDER_1.TUBE_SECTION_3_L1, FIFTH_STEP_DONE := "DB17000_MAINTENANCE_GLOBAL_VARIABLES".ACTION_DONE.POWDER.UNIT_2.FEEDER_1.TUBE_SECTION_3_L2, SIXTH_STEP_DONE := "DB17000_MAINTENANCE_GLOBAL_VARIABLES".ACTION_DONE.POWDER.UNIT_2.FEEDER_2.TUBE_SECTION_3_L2, SEVENTH_STEP_DONE := 0, FIRST_OPERATOR_HELP => "DB17100_MAINTENANCE_OPERATOR_HELP".OPERATOR_HELP[26], SECOND_OPERATOR_HELP => "DB17100_MAINTENANCE_OPERATOR_HELP".OPERATOR_HELP[27], THRID_OPERATOR_HELP => "DB17100_MAINTENANCE_OPERATOR_HELP".OPERATOR_HELP[28], FOURTH_OPERATOR_HELP => "DB17100_MAINTENANCE_OPERATOR_HELP".OPERATOR_HELP[48], FIFTH_OPERATOR_HELP => "DB17100_MAINTENANCE_OPERATOR_HELP".OPERATOR_HELP[50], SIXTH_OPERATOR_HELP => "DB17100_MAINTENANCE_OPERATOR_HELP".OPERATOR_HELP[56], SEVENTH_OPERATOR_HELP => #NULL, MAINTENANCE_IN_PROGRESS => "DB17200_MAINTENANCE_SEQUENCE".MAINTENANCE_IN_PROGRESS[11])
   END_RUNG
   // the same network as SCL:
   "FC17900_MAINTENANCE_SEQUENCE"(REQUEST := 0,
                           NUMBER_STEPS := 6,
                           FIRST_STEP_DONE := "DB17000_MAINTENANCE_GLOBAL_VARIABLES".ACTION_DONE.POWDER.UNIT_2.GENERAL.POWDER_TUBE_SECTION_4,
                           SECOND_STEP_DONE := "DB17000_MAINTENANCE_GLOBAL_VARIABLES".ACTION_DONE.POWDER.UNIT_2.GENERAL.POWDER_TUBE_SECTION_5,
                           THRID_STEP_DONE := "DB17000_MAINTENANCE_GLOBAL_VARIABLES".ACTION_DONE.POWDER.UNIT_2.GENERAL.RIGID_TUBE_OF_SPLITTER,
                           FOURTH_STEP_DONE := "DB17000_MAINTENANCE_GLOBAL_VARIABLES".ACTION_DONE.POWDER.UNIT_2.FEEDER_1.TUBE_SECTION_3_L1,
                           FIFTH_STEP_DONE := "DB17000_MAINTENANCE_GLOBAL_VARIABLES".ACTION_DONE.POWDER.UNIT_2.FEEDER_1.TUBE_SECTION_3_L2,
                           SIXTH_STEP_DONE := "DB17000_MAINTENANCE_GLOBAL_VARIABLES".ACTION_DONE.POWDER.UNIT_2.FEEDER_2.TUBE_SECTION_3_L2,
                           SEVENTH_STEP_DONE := 0,
                           FIRST_OPERATOR_HELP => "DB17100_MAINTENANCE_OPERATOR_HELP".OPERATOR_HELP[26],
                           SECOND_OPERATOR_HELP => "DB17100_MAINTENANCE_OPERATOR_HELP".OPERATOR_HELP[27],
                           THRID_OPERATOR_HELP => "DB17100_MAINTENANCE_OPERATOR_HELP".OPERATOR_HELP[28],
                           FOURTH_OPERATOR_HELP => "DB17100_MAINTENANCE_OPERATOR_HELP".OPERATOR_HELP[48],
                           FIFTH_OPERATOR_HELP => "DB17100_MAINTENANCE_OPERATOR_HELP".OPERATOR_HELP[50],
                           SIXTH_OPERATOR_HELP => "DB17100_MAINTENANCE_OPERATOR_HELP".OPERATOR_HELP[56],
                           SEVENTH_OPERATOR_HELP => #NULL,
                           MAINTENANCE_IN_PROGRESS => "DB17200_MAINTENANCE_SEQUENCE".MAINTENANCE_IN_PROGRESS[11]);
END_REGION

REGION Network 16: FEEDER LEAK
   RUNG wire#powerrail
      "FC17900_MAINTENANCE_SEQUENCE"(REQUEST := 0, NUMBER_STEPS := 5, FIRST_STEP_DONE := "DB17000_MAINTENANCE_GLOBAL_VARIABLES".ACTION_DONE.POWDER.UNIT_1.FEEDER_1.HOPPER_L1, SECOND_STEP_DONE := "DB17000_MAINTENANCE_GLOBAL_VARIABLES".ACTION_DONE.POWDER.UNIT_1.FEEDER_1.HOPPER_L2, THRID_STEP_DONE := "DB17000_MAINTENANCE_GLOBAL_VARIABLES".ACTION_DONE.POWDER.UNIT_2.FEEDER_1.HOPPER_L1, FOURTH_STEP_DONE := "DB17000_MAINTENANCE_GLOBAL_VARIABLES".ACTION_DONE.POWDER.UNIT_2.FEEDER_1.HOPPER_L2, FIFTH_STEP_DONE := "DB17000_MAINTENANCE_GLOBAL_VARIABLES".ACTION_DONE.POWDER.UNIT_2.FEEDER_2.HOPPER_L2, SIXTH_STEP_DONE := 0, SEVENTH_STEP_DONE := 0, FIRST_OPERATOR_HELP => "DB17100_MAINTENANCE_OPERATOR_HELP".OPERATOR_HELP[18], SECOND_OPERATOR_HELP => "DB17100_MAINTENANCE_OPERATOR_HELP".OPERATOR_HELP[20], THRID_OPERATOR_HELP => "DB17100_MAINTENANCE_OPERATOR_HELP".OPERATOR_HELP[47], FOURTH_OPERATOR_HELP => "DB17100_MAINTENANCE_OPERATOR_HELP".OPERATOR_HELP[49], FIFTH_OPERATOR_HELP => "DB17100_MAINTENANCE_OPERATOR_HELP".OPERATOR_HELP[55], SIXTH_OPERATOR_HELP => #NULL, SEVENTH_OPERATOR_HELP => #NULL, MAINTENANCE_IN_PROGRESS => "DB17200_MAINTENANCE_SEQUENCE".MAINTENANCE_IN_PROGRESS[12])
   END_RUNG
   // the same network as SCL:
   "FC17900_MAINTENANCE_SEQUENCE"(REQUEST := 0,
                           NUMBER_STEPS := 5,
                           FIRST_STEP_DONE := "DB17000_MAINTENANCE_GLOBAL_VARIABLES".ACTION_DONE.POWDER.UNIT_1.FEEDER_1.HOPPER_L1,
                           SECOND_STEP_DONE := "DB17000_MAINTENANCE_GLOBAL_VARIABLES".ACTION_DONE.POWDER.UNIT_1.FEEDER_1.HOPPER_L2,
                           THRID_STEP_DONE := "DB17000_MAINTENANCE_GLOBAL_VARIABLES".ACTION_DONE.POWDER.UNIT_2.FEEDER_1.HOPPER_L1,
                           FOURTH_STEP_DONE := "DB17000_MAINTENANCE_GLOBAL_VARIABLES".ACTION_DONE.POWDER.UNIT_2.FEEDER_1.HOPPER_L2,
                           FIFTH_STEP_DONE := "DB17000_MAINTENANCE_GLOBAL_VARIABLES".ACTION_DONE.POWDER.UNIT_2.FEEDER_2.HOPPER_L2,
                           SIXTH_STEP_DONE := 0,
                           SEVENTH_STEP_DONE := 0,
                           FIRST_OPERATOR_HELP => "DB17100_MAINTENANCE_OPERATOR_HELP".OPERATOR_HELP[18],
                           SECOND_OPERATOR_HELP => "DB17100_MAINTENANCE_OPERATOR_HELP".OPERATOR_HELP[20],
                           THRID_OPERATOR_HELP => "DB17100_MAINTENANCE_OPERATOR_HELP".OPERATOR_HELP[47],
                           FOURTH_OPERATOR_HELP => "DB17100_MAINTENANCE_OPERATOR_HELP".OPERATOR_HELP[49],
                           FIFTH_OPERATOR_HELP => "DB17100_MAINTENANCE_OPERATOR_HELP".OPERATOR_HELP[55],
                           SIXTH_OPERATOR_HELP => #NULL,
                           SEVENTH_OPERATOR_HELP => #NULL,
                           MAINTENANCE_IN_PROGRESS => "DB17200_MAINTENANCE_SEQUENCE".MAINTENANCE_IN_PROGRESS[12]);
END_REGION

REGION Network 17: HOOKED POWDER LINE UNIT 1
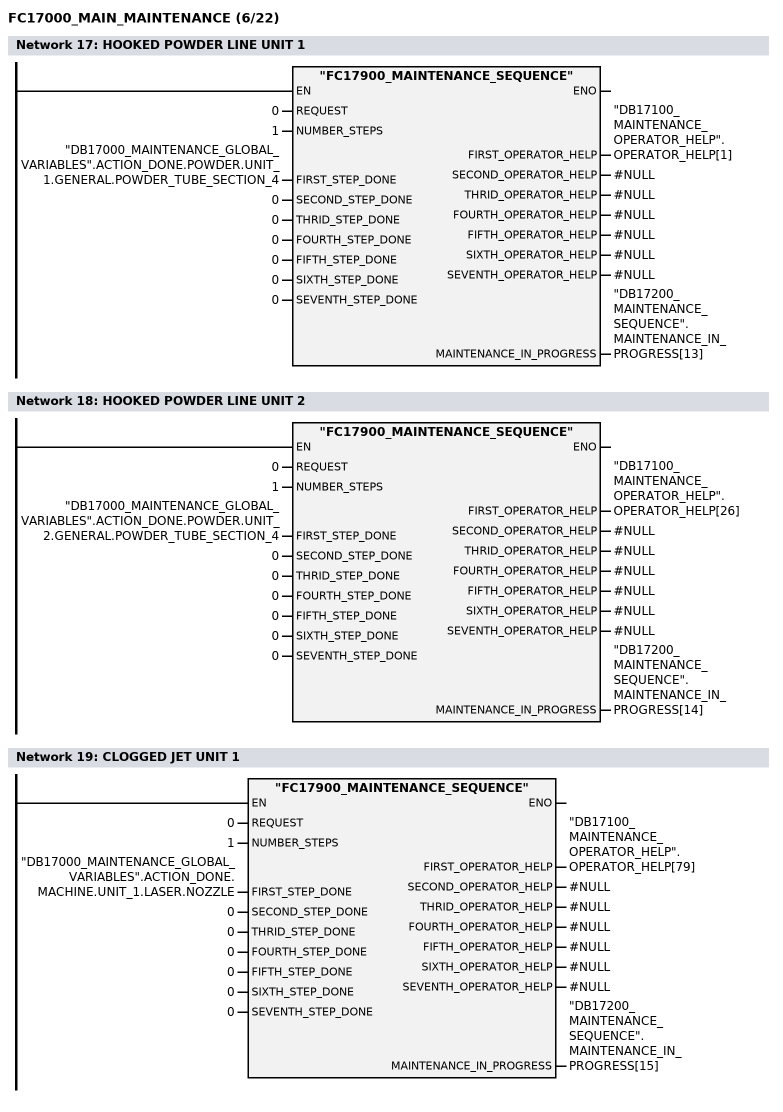
   RUNG wire#powerrail
      "FC17900_MAINTENANCE_SEQUENCE"(REQUEST := 0, NUMBER_STEPS := 1, FIRST_STEP_DONE := "DB17000_MAINTENANCE_GLOBAL_VARIABLES".ACTION_DONE.POWDER.UNIT_1.GENERAL.POWDER_TUBE_SECTION_4, SECOND_STEP_DONE := 0, THRID_STEP_DONE := 0, FOURTH_STEP_DONE := 0, FIFTH_STEP_DONE := 0, SIXTH_STEP_DONE := 0, SEVENTH_STEP_DONE := 0, FIRST_OPERATOR_HELP => "DB17100_MAINTENANCE_OPERATOR_HELP".OPERATOR_HELP[1], SECOND_OPERATOR_HELP => #NULL, THRID_OPERATOR_HELP => #NULL, FOURTH_OPERATOR_HELP => #NULL, FIFTH_OPERATOR_HELP => #NULL, SIXTH_OPERATOR_HELP => #NULL, SEVENTH_OPERATOR_HELP => #NULL, MAINTENANCE_IN_PROGRESS => "DB17200_MAINTENANCE_SEQUENCE".MAINTENANCE_IN_PROGRESS[13])
   END_RUNG
   // the same network as SCL:
   "FC17900_MAINTENANCE_SEQUENCE"(REQUEST := 0,
                           NUMBER_STEPS := 1,
                           FIRST_STEP_DONE := "DB17000_MAINTENANCE_GLOBAL_VARIABLES".ACTION_DONE.POWDER.UNIT_1.GENERAL.POWDER_TUBE_SECTION_4,
                           SECOND_STEP_DONE := 0,
                           THRID_STEP_DONE := 0,
                           FOURTH_STEP_DONE := 0,
                           FIFTH_STEP_DONE := 0,
                           SIXTH_STEP_DONE := 0,
                           SEVENTH_STEP_DONE := 0,
                           FIRST_OPERATOR_HELP => "DB17100_MAINTENANCE_OPERATOR_HELP".OPERATOR_HELP[1],
                           SECOND_OPERATOR_HELP => #NULL,
                           THRID_OPERATOR_HELP => #NULL,
                           FOURTH_OPERATOR_HELP => #NULL,
                           FIFTH_OPERATOR_HELP => #NULL,
                           SIXTH_OPERATOR_HELP => #NULL,
                           SEVENTH_OPERATOR_HELP => #NULL,
                           MAINTENANCE_IN_PROGRESS => "DB17200_MAINTENANCE_SEQUENCE".MAINTENANCE_IN_PROGRESS[13]);
END_REGION

REGION Network 18: HOOKED POWDER LINE UNIT 2
   RUNG wire#powerrail
      "FC17900_MAINTENANCE_SEQUENCE"(REQUEST := 0, NUMBER_STEPS := 1, FIRST_STEP_DONE := "DB17000_MAINTENANCE_GLOBAL_VARIABLES".ACTION_DONE.POWDER.UNIT_2.GENERAL.POWDER_TUBE_SECTION_4, SECOND_STEP_DONE := 0, THRID_STEP_DONE := 0, FOURTH_STEP_DONE := 0, FIFTH_STEP_DONE := 0, SIXTH_STEP_DONE := 0, SEVENTH_STEP_DONE := 0, FIRST_OPERATOR_HELP => "DB17100_MAINTENANCE_OPERATOR_HELP".OPERATOR_HELP[26], SECOND_OPERATOR_HELP => #NULL, THRID_OPERATOR_HELP => #NULL, FOURTH_OPERATOR_HELP => #NULL, FIFTH_OPERATOR_HELP => #NULL, SIXTH_OPERATOR_HELP => #NULL, SEVENTH_OPERATOR_HELP => #NULL, MAINTENANCE_IN_PROGRESS => "DB17200_MAINTENANCE_SEQUENCE".MAINTENANCE_IN_PROGRESS[14])
   END_RUNG
   // the same network as SCL:
   "FC17900_MAINTENANCE_SEQUENCE"(REQUEST := 0,
                           NUMBER_STEPS := 1,
                           FIRST_STEP_DONE := "DB17000_MAINTENANCE_GLOBAL_VARIABLES".ACTION_DONE.POWDER.UNIT_2.GENERAL.POWDER_TUBE_SECTION_4,
                           SECOND_STEP_DONE := 0,
                           THRID_STEP_DONE := 0,
                           FOURTH_STEP_DONE := 0,
                           FIFTH_STEP_DONE := 0,
                           SIXTH_STEP_DONE := 0,
                           SEVENTH_STEP_DONE := 0,
                           FIRST_OPERATOR_HELP => "DB17100_MAINTENANCE_OPERATOR_HELP".OPERATOR_HELP[26],
                           SECOND_OPERATOR_HELP => #NULL,
                           THRID_OPERATOR_HELP => #NULL,
                           FOURTH_OPERATOR_HELP => #NULL,
                           FIFTH_OPERATOR_HELP => #NULL,
                           SIXTH_OPERATOR_HELP => #NULL,
                           SEVENTH_OPERATOR_HELP => #NULL,
                           MAINTENANCE_IN_PROGRESS => "DB17200_MAINTENANCE_SEQUENCE".MAINTENANCE_IN_PROGRESS[14]);
END_REGION

REGION Network 19: CLOGGED JET UNIT 1
   RUNG wire#powerrail
      "FC17900_MAINTENANCE_SEQUENCE"(REQUEST := 0, NUMBER_STEPS := 1, FIRST_STEP_DONE := "DB17000_MAINTENANCE_GLOBAL_VARIABLES".ACTION_DONE.MACHINE.UNIT_1.LASER.NOZZLE, SECOND_STEP_DONE := 0, THRID_STEP_DONE := 0, FOURTH_STEP_DONE := 0, FIFTH_STEP_DONE := 0, SIXTH_STEP_DONE := 0, SEVENTH_STEP_DONE := 0, FIRST_OPERATOR_HELP => "DB17100_MAINTENANCE_OPERATOR_HELP".OPERATOR_HELP[79], SECOND_OPERATOR_HELP => #NULL, THRID_OPERATOR_HELP => #NULL, FOURTH_OPERATOR_HELP => #NULL, FIFTH_OPERATOR_HELP => #NULL, SIXTH_OPERATOR_HELP => #NULL, SEVENTH_OPERATOR_HELP => #NULL, MAINTENANCE_IN_PROGRESS => "DB17200_MAINTENANCE_SEQUENCE".MAINTENANCE_IN_PROGRESS[15])
   END_RUNG
   // the same network as SCL:
   "FC17900_MAINTENANCE_SEQUENCE"(REQUEST := 0,
                           NUMBER_STEPS := 1,
                           FIRST_STEP_DONE := "DB17000_MAINTENANCE_GLOBAL_VARIABLES".ACTION_DONE.MACHINE.UNIT_1.LASER.NOZZLE,
                           SECOND_STEP_DONE := 0,
                           THRID_STEP_DONE := 0,
                           FOURTH_STEP_DONE := 0,
                           FIFTH_STEP_DONE := 0,
                           SIXTH_STEP_DONE := 0,
                           SEVENTH_STEP_DONE := 0,
                           FIRST_OPERATOR_HELP => "DB17100_MAINTENANCE_OPERATOR_HELP".OPERATOR_HELP[79],
                           SECOND_OPERATOR_HELP => #NULL,
                           THRID_OPERATOR_HELP => #NULL,
                           FOURTH_OPERATOR_HELP => #NULL,
                           FIFTH_OPERATOR_HELP => #NULL,
                           SIXTH_OPERATOR_HELP => #NULL,
                           SEVENTH_OPERATOR_HELP => #NULL,
                           MAINTENANCE_IN_PROGRESS => "DB17200_MAINTENANCE_SEQUENCE".MAINTENANCE_IN_PROGRESS[15]);
END_REGION

REGION Network 20: CLOGGED JET UNIT 2
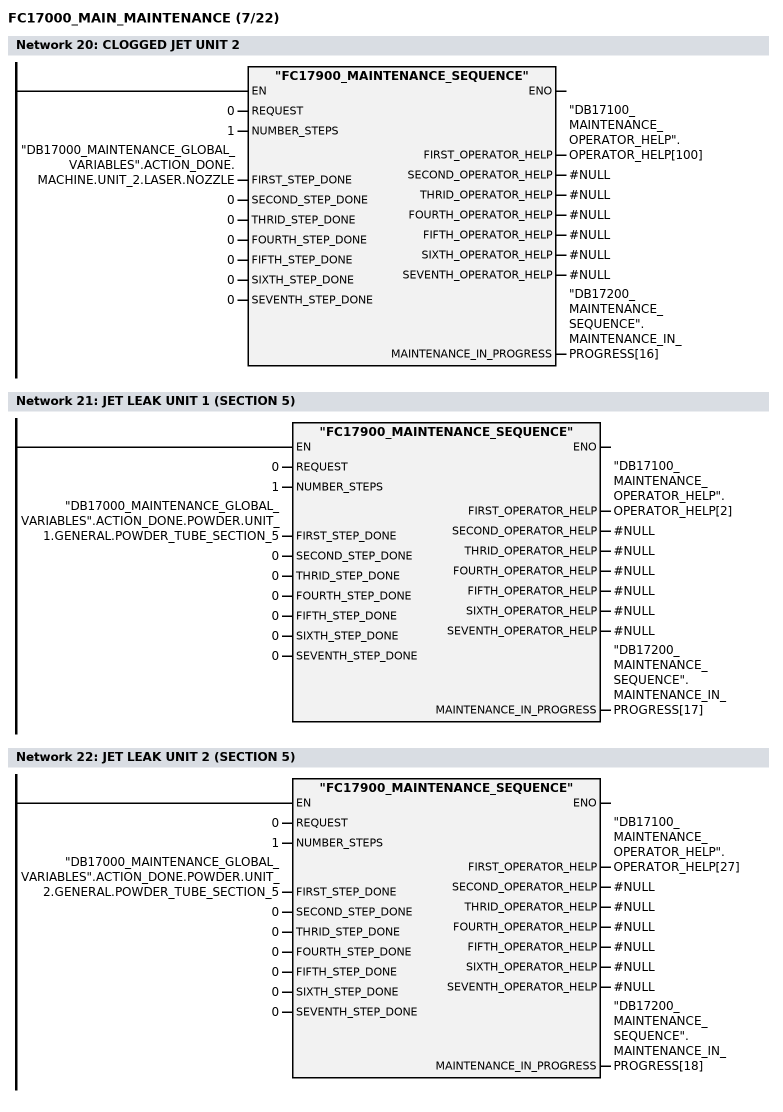
   RUNG wire#powerrail
      "FC17900_MAINTENANCE_SEQUENCE"(REQUEST := 0, NUMBER_STEPS := 1, FIRST_STEP_DONE := "DB17000_MAINTENANCE_GLOBAL_VARIABLES".ACTION_DONE.MACHINE.UNIT_2.LASER.NOZZLE, SECOND_STEP_DONE := 0, THRID_STEP_DONE := 0, FOURTH_STEP_DONE := 0, FIFTH_STEP_DONE := 0, SIXTH_STEP_DONE := 0, SEVENTH_STEP_DONE := 0, FIRST_OPERATOR_HELP => "DB17100_MAINTENANCE_OPERATOR_HELP".OPERATOR_HELP[100], SECOND_OPERATOR_HELP => #NULL, THRID_OPERATOR_HELP => #NULL, FOURTH_OPERATOR_HELP => #NULL, FIFTH_OPERATOR_HELP => #NULL, SIXTH_OPERATOR_HELP => #NULL, SEVENTH_OPERATOR_HELP => #NULL, MAINTENANCE_IN_PROGRESS => "DB17200_MAINTENANCE_SEQUENCE".MAINTENANCE_IN_PROGRESS[16])
   END_RUNG
   // the same network as SCL:
   "FC17900_MAINTENANCE_SEQUENCE"(REQUEST := 0,
                           NUMBER_STEPS := 1,
                           FIRST_STEP_DONE := "DB17000_MAINTENANCE_GLOBAL_VARIABLES".ACTION_DONE.MACHINE.UNIT_2.LASER.NOZZLE,
                           SECOND_STEP_DONE := 0,
                           THRID_STEP_DONE := 0,
                           FOURTH_STEP_DONE := 0,
                           FIFTH_STEP_DONE := 0,
                           SIXTH_STEP_DONE := 0,
                           SEVENTH_STEP_DONE := 0,
                           FIRST_OPERATOR_HELP => "DB17100_MAINTENANCE_OPERATOR_HELP".OPERATOR_HELP[100],
                           SECOND_OPERATOR_HELP => #NULL,
                           THRID_OPERATOR_HELP => #NULL,
                           FOURTH_OPERATOR_HELP => #NULL,
                           FIFTH_OPERATOR_HELP => #NULL,
                           SIXTH_OPERATOR_HELP => #NULL,
                           SEVENTH_OPERATOR_HELP => #NULL,
                           MAINTENANCE_IN_PROGRESS => "DB17200_MAINTENANCE_SEQUENCE".MAINTENANCE_IN_PROGRESS[16]);
END_REGION

REGION Network 21: JET LEAK UNIT 1 (SECTION 5)
   RUNG wire#powerrail
      "FC17900_MAINTENANCE_SEQUENCE"(REQUEST := 0, NUMBER_STEPS := 1, FIRST_STEP_DONE := "DB17000_MAINTENANCE_GLOBAL_VARIABLES".ACTION_DONE.POWDER.UNIT_1.GENERAL.POWDER_TUBE_SECTION_5, SECOND_STEP_DONE := 0, THRID_STEP_DONE := 0, FOURTH_STEP_DONE := 0, FIFTH_STEP_DONE := 0, SIXTH_STEP_DONE := 0, SEVENTH_STEP_DONE := 0, FIRST_OPERATOR_HELP => "DB17100_MAINTENANCE_OPERATOR_HELP".OPERATOR_HELP[2], SECOND_OPERATOR_HELP => #NULL, THRID_OPERATOR_HELP => #NULL, FOURTH_OPERATOR_HELP => #NULL, FIFTH_OPERATOR_HELP => #NULL, SIXTH_OPERATOR_HELP => #NULL, SEVENTH_OPERATOR_HELP => #NULL, MAINTENANCE_IN_PROGRESS => "DB17200_MAINTENANCE_SEQUENCE".MAINTENANCE_IN_PROGRESS[17])
   END_RUNG
   // the same network as SCL:
   "FC17900_MAINTENANCE_SEQUENCE"(REQUEST := 0,
                           NUMBER_STEPS := 1,
                           FIRST_STEP_DONE := "DB17000_MAINTENANCE_GLOBAL_VARIABLES".ACTION_DONE.POWDER.UNIT_1.GENERAL.POWDER_TUBE_SECTION_5,
                           SECOND_STEP_DONE := 0,
                           THRID_STEP_DONE := 0,
                           FOURTH_STEP_DONE := 0,
                           FIFTH_STEP_DONE := 0,
                           SIXTH_STEP_DONE := 0,
                           SEVENTH_STEP_DONE := 0,
                           FIRST_OPERATOR_HELP => "DB17100_MAINTENANCE_OPERATOR_HELP".OPERATOR_HELP[2],
                           SECOND_OPERATOR_HELP => #NULL,
                           THRID_OPERATOR_HELP => #NULL,
                           FOURTH_OPERATOR_HELP => #NULL,
                           FIFTH_OPERATOR_HELP => #NULL,
                           SIXTH_OPERATOR_HELP => #NULL,
                           SEVENTH_OPERATOR_HELP => #NULL,
                           MAINTENANCE_IN_PROGRESS => "DB17200_MAINTENANCE_SEQUENCE".MAINTENANCE_IN_PROGRESS[17]);
END_REGION

REGION Network 22: JET LEAK UNIT 2 (SECTION 5)
   RUNG wire#powerrail
      "FC17900_MAINTENANCE_SEQUENCE"(REQUEST := 0, NUMBER_STEPS := 1, FIRST_STEP_DONE := "DB17000_MAINTENANCE_GLOBAL_VARIABLES".ACTION_DONE.POWDER.UNIT_2.GENERAL.POWDER_TUBE_SECTION_5, SECOND_STEP_DONE := 0, THRID_STEP_DONE := 0, FOURTH_STEP_DONE := 0, FIFTH_STEP_DONE := 0, SIXTH_STEP_DONE := 0, SEVENTH_STEP_DONE := 0, FIRST_OPERATOR_HELP => "DB17100_MAINTENANCE_OPERATOR_HELP".OPERATOR_HELP[27], SECOND_OPERATOR_HELP => #NULL, THRID_OPERATOR_HELP => #NULL, FOURTH_OPERATOR_HELP => #NULL, FIFTH_OPERATOR_HELP => #NULL, SIXTH_OPERATOR_HELP => #NULL, SEVENTH_OPERATOR_HELP => #NULL, MAINTENANCE_IN_PROGRESS => "DB17200_MAINTENANCE_SEQUENCE".MAINTENANCE_IN_PROGRESS[18])
   END_RUNG
   // the same network as SCL:
   "FC17900_MAINTENANCE_SEQUENCE"(REQUEST := 0,
                           NUMBER_STEPS := 1,
                           FIRST_STEP_DONE := "DB17000_MAINTENANCE_GLOBAL_VARIABLES".ACTION_DONE.POWDER.UNIT_2.GENERAL.POWDER_TUBE_SECTION_5,
                           SECOND_STEP_DONE := 0,
                           THRID_STEP_DONE := 0,
                           FOURTH_STEP_DONE := 0,
                           FIFTH_STEP_DONE := 0,
                           SIXTH_STEP_DONE := 0,
                           SEVENTH_STEP_DONE := 0,
                           FIRST_OPERATOR_HELP => "DB17100_MAINTENANCE_OPERATOR_HELP".OPERATOR_HELP[27],
                           SECOND_OPERATOR_HELP => #NULL,
                           THRID_OPERATOR_HELP => #NULL,
                           FOURTH_OPERATOR_HELP => #NULL,
                           FIFTH_OPERATOR_HELP => #NULL,
                           SIXTH_OPERATOR_HELP => #NULL,
                           SEVENTH_OPERATOR_HELP => #NULL,
                           MAINTENANCE_IN_PROGRESS => "DB17200_MAINTENANCE_SEQUENCE".MAINTENANCE_IN_PROGRESS[18]);
END_REGION

REGION Network 23: REJECTED PARTS UNIT 1
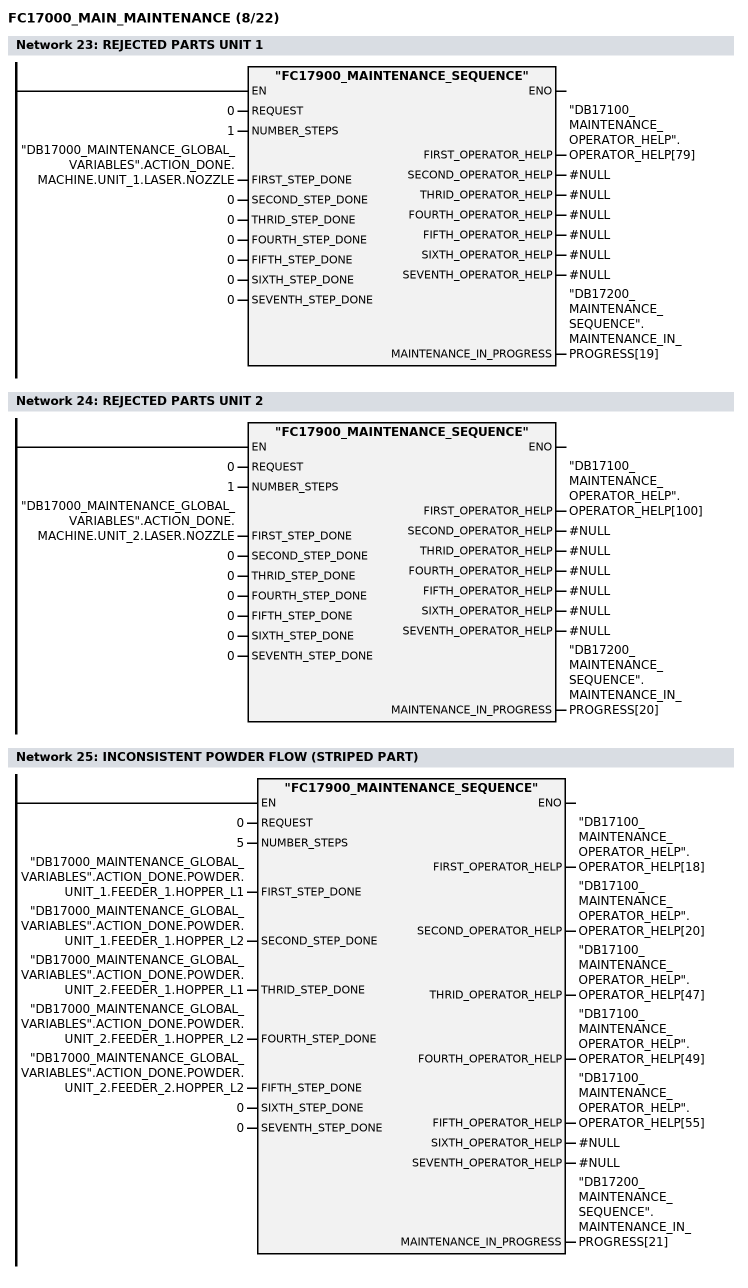
   RUNG wire#powerrail
      "FC17900_MAINTENANCE_SEQUENCE"(REQUEST := 0, NUMBER_STEPS := 1, FIRST_STEP_DONE := "DB17000_MAINTENANCE_GLOBAL_VARIABLES".ACTION_DONE.MACHINE.UNIT_1.LASER.NOZZLE, SECOND_STEP_DONE := 0, THRID_STEP_DONE := 0, FOURTH_STEP_DONE := 0, FIFTH_STEP_DONE := 0, SIXTH_STEP_DONE := 0, SEVENTH_STEP_DONE := 0, FIRST_OPERATOR_HELP => "DB17100_MAINTENANCE_OPERATOR_HELP".OPERATOR_HELP[79], SECOND_OPERATOR_HELP => #NULL, THRID_OPERATOR_HELP => #NULL, FOURTH_OPERATOR_HELP => #NULL, FIFTH_OPERATOR_HELP => #NULL, SIXTH_OPERATOR_HELP => #NULL, SEVENTH_OPERATOR_HELP => #NULL, MAINTENANCE_IN_PROGRESS => "DB17200_MAINTENANCE_SEQUENCE".MAINTENANCE_IN_PROGRESS[19])
   END_RUNG
   // the same network as SCL:
   "FC17900_MAINTENANCE_SEQUENCE"(REQUEST := 0,
                           NUMBER_STEPS := 1,
                           FIRST_STEP_DONE := "DB17000_MAINTENANCE_GLOBAL_VARIABLES".ACTION_DONE.MACHINE.UNIT_1.LASER.NOZZLE,
                           SECOND_STEP_DONE := 0,
                           THRID_STEP_DONE := 0,
                           FOURTH_STEP_DONE := 0,
                           FIFTH_STEP_DONE := 0,
                           SIXTH_STEP_DONE := 0,
                           SEVENTH_STEP_DONE := 0,
                           FIRST_OPERATOR_HELP => "DB17100_MAINTENANCE_OPERATOR_HELP".OPERATOR_HELP[79],
                           SECOND_OPERATOR_HELP => #NULL,
                           THRID_OPERATOR_HELP => #NULL,
                           FOURTH_OPERATOR_HELP => #NULL,
                           FIFTH_OPERATOR_HELP => #NULL,
                           SIXTH_OPERATOR_HELP => #NULL,
                           SEVENTH_OPERATOR_HELP => #NULL,
                           MAINTENANCE_IN_PROGRESS => "DB17200_MAINTENANCE_SEQUENCE".MAINTENANCE_IN_PROGRESS[19]);
END_REGION

REGION Network 24: REJECTED PARTS UNIT 2
   RUNG wire#powerrail
      "FC17900_MAINTENANCE_SEQUENCE"(REQUEST := 0, NUMBER_STEPS := 1, FIRST_STEP_DONE := "DB17000_MAINTENANCE_GLOBAL_VARIABLES".ACTION_DONE.MACHINE.UNIT_2.LASER.NOZZLE, SECOND_STEP_DONE := 0, THRID_STEP_DONE := 0, FOURTH_STEP_DONE := 0, FIFTH_STEP_DONE := 0, SIXTH_STEP_DONE := 0, SEVENTH_STEP_DONE := 0, FIRST_OPERATOR_HELP => "DB17100_MAINTENANCE_OPERATOR_HELP".OPERATOR_HELP[100], SECOND_OPERATOR_HELP => #NULL, THRID_OPERATOR_HELP => #NULL, FOURTH_OPERATOR_HELP => #NULL, FIFTH_OPERATOR_HELP => #NULL, SIXTH_OPERATOR_HELP => #NULL, SEVENTH_OPERATOR_HELP => #NULL, MAINTENANCE_IN_PROGRESS => "DB17200_MAINTENANCE_SEQUENCE".MAINTENANCE_IN_PROGRESS[20])
   END_RUNG
   // the same network as SCL:
   "FC17900_MAINTENANCE_SEQUENCE"(REQUEST := 0,
                           NUMBER_STEPS := 1,
                           FIRST_STEP_DONE := "DB17000_MAINTENANCE_GLOBAL_VARIABLES".ACTION_DONE.MACHINE.UNIT_2.LASER.NOZZLE,
                           SECOND_STEP_DONE := 0,
                           THRID_STEP_DONE := 0,
                           FOURTH_STEP_DONE := 0,
                           FIFTH_STEP_DONE := 0,
                           SIXTH_STEP_DONE := 0,
                           SEVENTH_STEP_DONE := 0,
                           FIRST_OPERATOR_HELP => "DB17100_MAINTENANCE_OPERATOR_HELP".OPERATOR_HELP[100],
                           SECOND_OPERATOR_HELP => #NULL,
                           THRID_OPERATOR_HELP => #NULL,
                           FOURTH_OPERATOR_HELP => #NULL,
                           FIFTH_OPERATOR_HELP => #NULL,
                           SIXTH_OPERATOR_HELP => #NULL,
                           SEVENTH_OPERATOR_HELP => #NULL,
                           MAINTENANCE_IN_PROGRESS => "DB17200_MAINTENANCE_SEQUENCE".MAINTENANCE_IN_PROGRESS[20]);
END_REGION

REGION Network 25: INCONSISTENT POWDER FLOW (STRIPED PART)
   RUNG wire#powerrail
      "FC17900_MAINTENANCE_SEQUENCE"(REQUEST := 0, NUMBER_STEPS := 5, FIRST_STEP_DONE := "DB17000_MAINTENANCE_GLOBAL_VARIABLES".ACTION_DONE.POWDER.UNIT_1.FEEDER_1.HOPPER_L1, SECOND_STEP_DONE := "DB17000_MAINTENANCE_GLOBAL_VARIABLES".ACTION_DONE.POWDER.UNIT_1.FEEDER_1.HOPPER_L2, THRID_STEP_DONE := "DB17000_MAINTENANCE_GLOBAL_VARIABLES".ACTION_DONE.POWDER.UNIT_2.FEEDER_1.HOPPER_L1, FOURTH_STEP_DONE := "DB17000_MAINTENANCE_GLOBAL_VARIABLES".ACTION_DONE.POWDER.UNIT_2.FEEDER_1.HOPPER_L2, FIFTH_STEP_DONE := "DB17000_MAINTENANCE_GLOBAL_VARIABLES".ACTION_DONE.POWDER.UNIT_2.FEEDER_2.HOPPER_L2, SIXTH_STEP_DONE := 0, SEVENTH_STEP_DONE := 0, FIRST_OPERATOR_HELP => "DB17100_MAINTENANCE_OPERATOR_HELP".OPERATOR_HELP[18], SECOND_OPERATOR_HELP => "DB17100_MAINTENANCE_OPERATOR_HELP".OPERATOR_HELP[20], THRID_OPERATOR_HELP => "DB17100_MAINTENANCE_OPERATOR_HELP".OPERATOR_HELP[47], FOURTH_OPERATOR_HELP => "DB17100_MAINTENANCE_OPERATOR_HELP".OPERATOR_HELP[49], FIFTH_OPERATOR_HELP => "DB17100_MAINTENANCE_OPERATOR_HELP".OPERATOR_HELP[55], SIXTH_OPERATOR_HELP => #NULL, SEVENTH_OPERATOR_HELP => #NULL, MAINTENANCE_IN_PROGRESS => "DB17200_MAINTENANCE_SEQUENCE".MAINTENANCE_IN_PROGRESS[21])
   END_RUNG
   // the same network as SCL:
   "FC17900_MAINTENANCE_SEQUENCE"(REQUEST := 0,
                           NUMBER_STEPS := 5,
                           FIRST_STEP_DONE := "DB17000_MAINTENANCE_GLOBAL_VARIABLES".ACTION_DONE.POWDER.UNIT_1.FEEDER_1.HOPPER_L1,
                           SECOND_STEP_DONE := "DB17000_MAINTENANCE_GLOBAL_VARIABLES".ACTION_DONE.POWDER.UNIT_1.FEEDER_1.HOPPER_L2,
                           THRID_STEP_DONE := "DB17000_MAINTENANCE_GLOBAL_VARIABLES".ACTION_DONE.POWDER.UNIT_2.FEEDER_1.HOPPER_L1,
                           FOURTH_STEP_DONE := "DB17000_MAINTENANCE_GLOBAL_VARIABLES".ACTION_DONE.POWDER.UNIT_2.FEEDER_1.HOPPER_L2,
                           FIFTH_STEP_DONE := "DB17000_MAINTENANCE_GLOBAL_VARIABLES".ACTION_DONE.POWDER.UNIT_2.FEEDER_2.HOPPER_L2,
                           SIXTH_STEP_DONE := 0,
                           SEVENTH_STEP_DONE := 0,
                           FIRST_OPERATOR_HELP => "DB17100_MAINTENANCE_OPERATOR_HELP".OPERATOR_HELP[18],
                           SECOND_OPERATOR_HELP => "DB17100_MAINTENANCE_OPERATOR_HELP".OPERATOR_HELP[20],
                           THRID_OPERATOR_HELP => "DB17100_MAINTENANCE_OPERATOR_HELP".OPERATOR_HELP[47],
                           FOURTH_OPERATOR_HELP => "DB17100_MAINTENANCE_OPERATOR_HELP".OPERATOR_HELP[49],
                           FIFTH_OPERATOR_HELP => "DB17100_MAINTENANCE_OPERATOR_HELP".OPERATOR_HELP[55],
                           SIXTH_OPERATOR_HELP => #NULL,
                           SEVENTH_OPERATOR_HELP => #NULL,
                           MAINTENANCE_IN_PROGRESS => "DB17200_MAINTENANCE_SEQUENCE".MAINTENANCE_IN_PROGRESS[21]);
END_REGION

REGION Network 26: LAYER SHRINKING UNIT 1
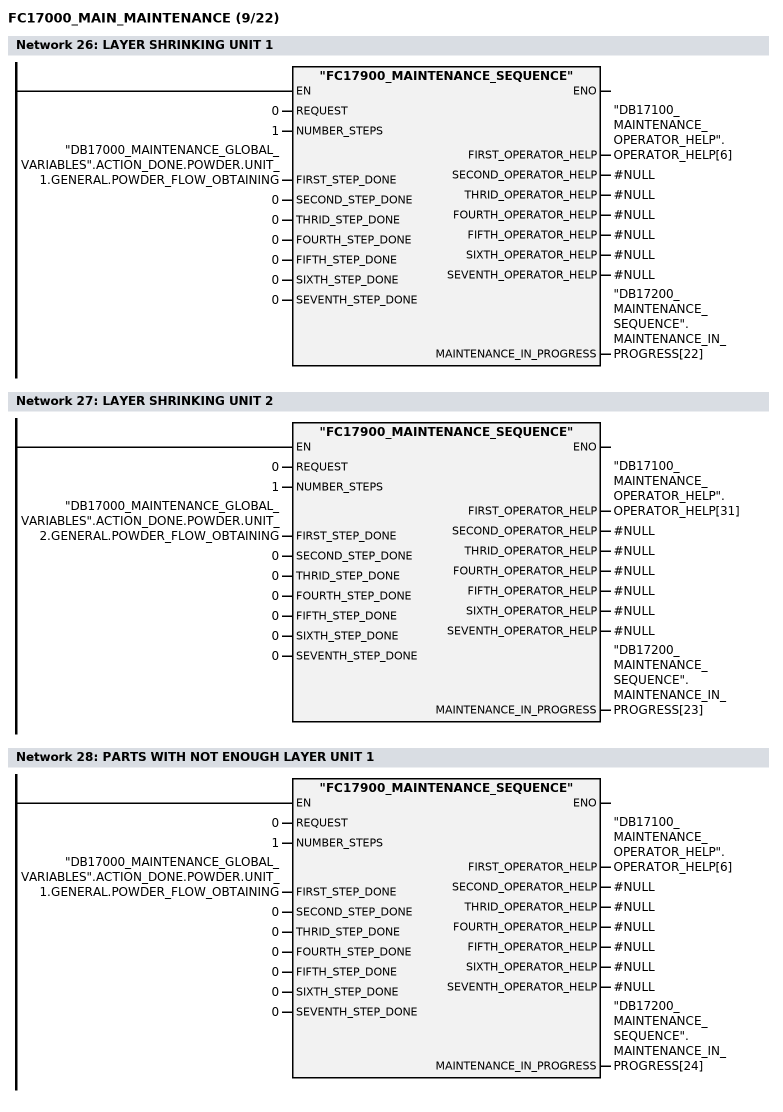
   RUNG wire#powerrail
      "FC17900_MAINTENANCE_SEQUENCE"(REQUEST := 0, NUMBER_STEPS := 1, FIRST_STEP_DONE := "DB17000_MAINTENANCE_GLOBAL_VARIABLES".ACTION_DONE.POWDER.UNIT_1.GENERAL.POWDER_FLOW_OBTAINING, SECOND_STEP_DONE := 0, THRID_STEP_DONE := 0, FOURTH_STEP_DONE := 0, FIFTH_STEP_DONE := 0, SIXTH_STEP_DONE := 0, SEVENTH_STEP_DONE := 0, FIRST_OPERATOR_HELP => "DB17100_MAINTENANCE_OPERATOR_HELP".OPERATOR_HELP[6], SECOND_OPERATOR_HELP => #NULL, THRID_OPERATOR_HELP => #NULL, FOURTH_OPERATOR_HELP => #NULL, FIFTH_OPERATOR_HELP => #NULL, SIXTH_OPERATOR_HELP => #NULL, SEVENTH_OPERATOR_HELP => #NULL, MAINTENANCE_IN_PROGRESS => "DB17200_MAINTENANCE_SEQUENCE".MAINTENANCE_IN_PROGRESS[22])
   END_RUNG
   // the same network as SCL:
   "FC17900_MAINTENANCE_SEQUENCE"(REQUEST := 0,
                           NUMBER_STEPS := 1,
                           FIRST_STEP_DONE := "DB17000_MAINTENANCE_GLOBAL_VARIABLES".ACTION_DONE.POWDER.UNIT_1.GENERAL.POWDER_FLOW_OBTAINING,
                           SECOND_STEP_DONE := 0,
                           THRID_STEP_DONE := 0,
                           FOURTH_STEP_DONE := 0,
                           FIFTH_STEP_DONE := 0,
                           SIXTH_STEP_DONE := 0,
                           SEVENTH_STEP_DONE := 0,
                           FIRST_OPERATOR_HELP => "DB17100_MAINTENANCE_OPERATOR_HELP".OPERATOR_HELP[6],
                           SECOND_OPERATOR_HELP => #NULL,
                           THRID_OPERATOR_HELP => #NULL,
                           FOURTH_OPERATOR_HELP => #NULL,
                           FIFTH_OPERATOR_HELP => #NULL,
                           SIXTH_OPERATOR_HELP => #NULL,
                           SEVENTH_OPERATOR_HELP => #NULL,
                           MAINTENANCE_IN_PROGRESS => "DB17200_MAINTENANCE_SEQUENCE".MAINTENANCE_IN_PROGRESS[22]);
END_REGION

REGION Network 27: LAYER SHRINKING UNIT 2
   RUNG wire#powerrail
      "FC17900_MAINTENANCE_SEQUENCE"(REQUEST := 0, NUMBER_STEPS := 1, FIRST_STEP_DONE := "DB17000_MAINTENANCE_GLOBAL_VARIABLES".ACTION_DONE.POWDER.UNIT_2.GENERAL.POWDER_FLOW_OBTAINING, SECOND_STEP_DONE := 0, THRID_STEP_DONE := 0, FOURTH_STEP_DONE := 0, FIFTH_STEP_DONE := 0, SIXTH_STEP_DONE := 0, SEVENTH_STEP_DONE := 0, FIRST_OPERATOR_HELP => "DB17100_MAINTENANCE_OPERATOR_HELP".OPERATOR_HELP[31], SECOND_OPERATOR_HELP => #NULL, THRID_OPERATOR_HELP => #NULL, FOURTH_OPERATOR_HELP => #NULL, FIFTH_OPERATOR_HELP => #NULL, SIXTH_OPERATOR_HELP => #NULL, SEVENTH_OPERATOR_HELP => #NULL, MAINTENANCE_IN_PROGRESS => "DB17200_MAINTENANCE_SEQUENCE".MAINTENANCE_IN_PROGRESS[23])
   END_RUNG
   // the same network as SCL:
   "FC17900_MAINTENANCE_SEQUENCE"(REQUEST := 0,
                           NUMBER_STEPS := 1,
                           FIRST_STEP_DONE := "DB17000_MAINTENANCE_GLOBAL_VARIABLES".ACTION_DONE.POWDER.UNIT_2.GENERAL.POWDER_FLOW_OBTAINING,
                           SECOND_STEP_DONE := 0,
                           THRID_STEP_DONE := 0,
                           FOURTH_STEP_DONE := 0,
                           FIFTH_STEP_DONE := 0,
                           SIXTH_STEP_DONE := 0,
                           SEVENTH_STEP_DONE := 0,
                           FIRST_OPERATOR_HELP => "DB17100_MAINTENANCE_OPERATOR_HELP".OPERATOR_HELP[31],
                           SECOND_OPERATOR_HELP => #NULL,
                           THRID_OPERATOR_HELP => #NULL,
                           FOURTH_OPERATOR_HELP => #NULL,
                           FIFTH_OPERATOR_HELP => #NULL,
                           SIXTH_OPERATOR_HELP => #NULL,
                           SEVENTH_OPERATOR_HELP => #NULL,
                           MAINTENANCE_IN_PROGRESS => "DB17200_MAINTENANCE_SEQUENCE".MAINTENANCE_IN_PROGRESS[23]);
END_REGION

REGION Network 28: PARTS WITH NOT ENOUGH LAYER UNIT 1
   RUNG wire#powerrail
      "FC17900_MAINTENANCE_SEQUENCE"(REQUEST := 0, NUMBER_STEPS := 1, FIRST_STEP_DONE := "DB17000_MAINTENANCE_GLOBAL_VARIABLES".ACTION_DONE.POWDER.UNIT_1.GENERAL.POWDER_FLOW_OBTAINING, SECOND_STEP_DONE := 0, THRID_STEP_DONE := 0, FOURTH_STEP_DONE := 0, FIFTH_STEP_DONE := 0, SIXTH_STEP_DONE := 0, SEVENTH_STEP_DONE := 0, FIRST_OPERATOR_HELP => "DB17100_MAINTENANCE_OPERATOR_HELP".OPERATOR_HELP[6], SECOND_OPERATOR_HELP => #NULL, THRID_OPERATOR_HELP => #NULL, FOURTH_OPERATOR_HELP => #NULL, FIFTH_OPERATOR_HELP => #NULL, SIXTH_OPERATOR_HELP => #NULL, SEVENTH_OPERATOR_HELP => #NULL, MAINTENANCE_IN_PROGRESS => "DB17200_MAINTENANCE_SEQUENCE".MAINTENANCE_IN_PROGRESS[24])
   END_RUNG
   // the same network as SCL:
   "FC17900_MAINTENANCE_SEQUENCE"(REQUEST := 0,
                           NUMBER_STEPS := 1,
                           FIRST_STEP_DONE := "DB17000_MAINTENANCE_GLOBAL_VARIABLES".ACTION_DONE.POWDER.UNIT_1.GENERAL.POWDER_FLOW_OBTAINING,
                           SECOND_STEP_DONE := 0,
                           THRID_STEP_DONE := 0,
                           FOURTH_STEP_DONE := 0,
                           FIFTH_STEP_DONE := 0,
                           SIXTH_STEP_DONE := 0,
                           SEVENTH_STEP_DONE := 0,
                           FIRST_OPERATOR_HELP => "DB17100_MAINTENANCE_OPERATOR_HELP".OPERATOR_HELP[6],
                           SECOND_OPERATOR_HELP => #NULL,
                           THRID_OPERATOR_HELP => #NULL,
                           FOURTH_OPERATOR_HELP => #NULL,
                           FIFTH_OPERATOR_HELP => #NULL,
                           SIXTH_OPERATOR_HELP => #NULL,
                           SEVENTH_OPERATOR_HELP => #NULL,
                           MAINTENANCE_IN_PROGRESS => "DB17200_MAINTENANCE_SEQUENCE".MAINTENANCE_IN_PROGRESS[24]);
END_REGION

REGION Network 29: PARTS WITH NOT ENOUGH LAYER UNIT 2
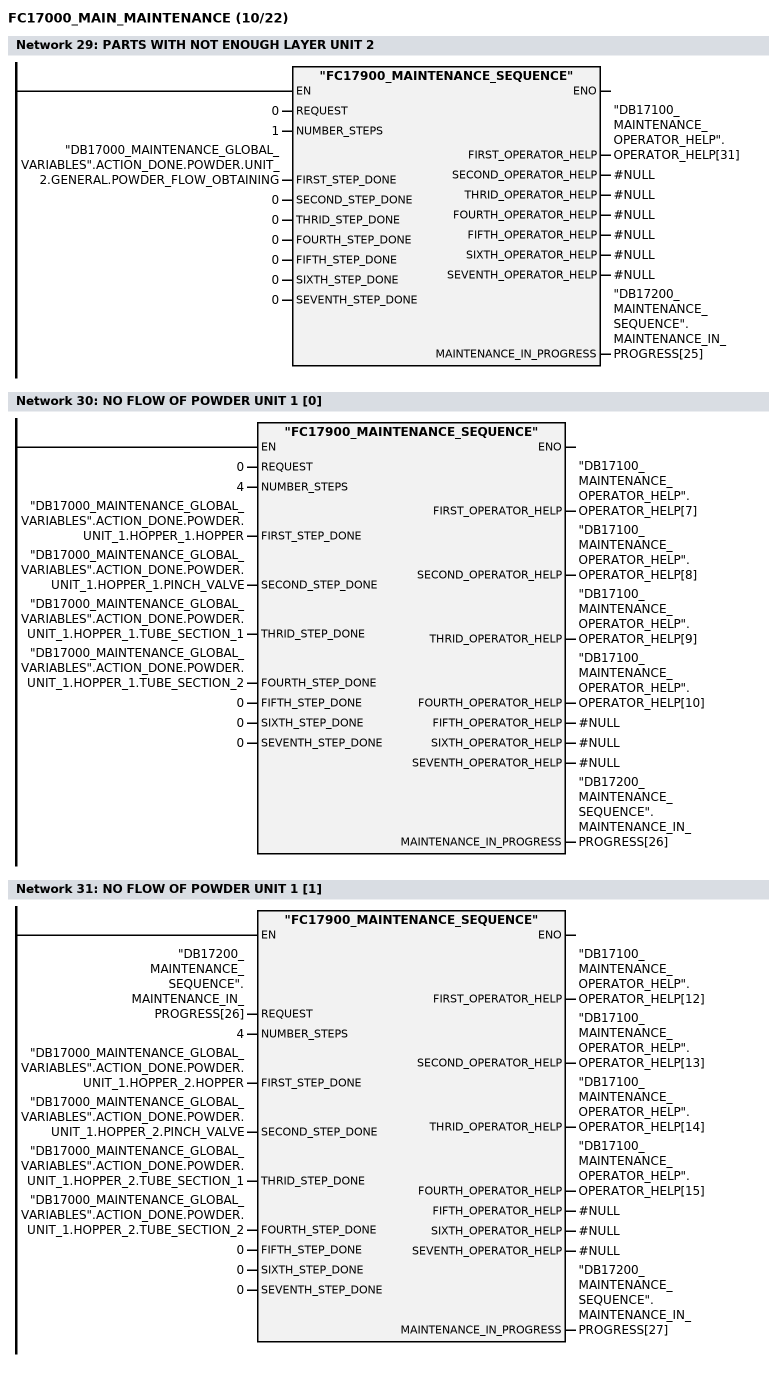
   RUNG wire#powerrail
      "FC17900_MAINTENANCE_SEQUENCE"(REQUEST := 0, NUMBER_STEPS := 1, FIRST_STEP_DONE := "DB17000_MAINTENANCE_GLOBAL_VARIABLES".ACTION_DONE.POWDER.UNIT_2.GENERAL.POWDER_FLOW_OBTAINING, SECOND_STEP_DONE := 0, THRID_STEP_DONE := 0, FOURTH_STEP_DONE := 0, FIFTH_STEP_DONE := 0, SIXTH_STEP_DONE := 0, SEVENTH_STEP_DONE := 0, FIRST_OPERATOR_HELP => "DB17100_MAINTENANCE_OPERATOR_HELP".OPERATOR_HELP[31], SECOND_OPERATOR_HELP => #NULL, THRID_OPERATOR_HELP => #NULL, FOURTH_OPERATOR_HELP => #NULL, FIFTH_OPERATOR_HELP => #NULL, SIXTH_OPERATOR_HELP => #NULL, SEVENTH_OPERATOR_HELP => #NULL, MAINTENANCE_IN_PROGRESS => "DB17200_MAINTENANCE_SEQUENCE".MAINTENANCE_IN_PROGRESS[25])
   END_RUNG
   // the same network as SCL:
   "FC17900_MAINTENANCE_SEQUENCE"(REQUEST := 0,
                           NUMBER_STEPS := 1,
                           FIRST_STEP_DONE := "DB17000_MAINTENANCE_GLOBAL_VARIABLES".ACTION_DONE.POWDER.UNIT_2.GENERAL.POWDER_FLOW_OBTAINING,
                           SECOND_STEP_DONE := 0,
                           THRID_STEP_DONE := 0,
                           FOURTH_STEP_DONE := 0,
                           FIFTH_STEP_DONE := 0,
                           SIXTH_STEP_DONE := 0,
                           SEVENTH_STEP_DONE := 0,
                           FIRST_OPERATOR_HELP => "DB17100_MAINTENANCE_OPERATOR_HELP".OPERATOR_HELP[31],
                           SECOND_OPERATOR_HELP => #NULL,
                           THRID_OPERATOR_HELP => #NULL,
                           FOURTH_OPERATOR_HELP => #NULL,
                           FIFTH_OPERATOR_HELP => #NULL,
                           SIXTH_OPERATOR_HELP => #NULL,
                           SEVENTH_OPERATOR_HELP => #NULL,
                           MAINTENANCE_IN_PROGRESS => "DB17200_MAINTENANCE_SEQUENCE".MAINTENANCE_IN_PROGRESS[25]);
END_REGION

REGION Network 30: NO FLOW OF POWDER UNIT 1 [0]
   RUNG wire#powerrail
      "FC17900_MAINTENANCE_SEQUENCE"(REQUEST := 0, NUMBER_STEPS := 4, FIRST_STEP_DONE := "DB17000_MAINTENANCE_GLOBAL_VARIABLES".ACTION_DONE.POWDER.UNIT_1.HOPPER_1.HOPPER, SECOND_STEP_DONE := "DB17000_MAINTENANCE_GLOBAL_VARIABLES".ACTION_DONE.POWDER.UNIT_1.HOPPER_1.PINCH_VALVE, THRID_STEP_DONE := "DB17000_MAINTENANCE_GLOBAL_VARIABLES".ACTION_DONE.POWDER.UNIT_1.HOPPER_1.TUBE_SECTION_1, FOURTH_STEP_DONE := "DB17000_MAINTENANCE_GLOBAL_VARIABLES".ACTION_DONE.POWDER.UNIT_1.HOPPER_1.TUBE_SECTION_2, FIFTH_STEP_DONE := 0, SIXTH_STEP_DONE := 0, SEVENTH_STEP_DONE := 0, FIRST_OPERATOR_HELP => "DB17100_MAINTENANCE_OPERATOR_HELP".OPERATOR_HELP[7], SECOND_OPERATOR_HELP => "DB17100_MAINTENANCE_OPERATOR_HELP".OPERATOR_HELP[8], THRID_OPERATOR_HELP => "DB17100_MAINTENANCE_OPERATOR_HELP".OPERATOR_HELP[9], FOURTH_OPERATOR_HELP => "DB17100_MAINTENANCE_OPERATOR_HELP".OPERATOR_HELP[10], FIFTH_OPERATOR_HELP => #NULL, SIXTH_OPERATOR_HELP => #NULL, SEVENTH_OPERATOR_HELP => #NULL, MAINTENANCE_IN_PROGRESS => "DB17200_MAINTENANCE_SEQUENCE".MAINTENANCE_IN_PROGRESS[26])
   END_RUNG
   // the same network as SCL:
   "FC17900_MAINTENANCE_SEQUENCE"(REQUEST := 0,
                           NUMBER_STEPS := 4,
                           FIRST_STEP_DONE := "DB17000_MAINTENANCE_GLOBAL_VARIABLES".ACTION_DONE.POWDER.UNIT_1.HOPPER_1.HOPPER,
                           SECOND_STEP_DONE := "DB17000_MAINTENANCE_GLOBAL_VARIABLES".ACTION_DONE.POWDER.UNIT_1.HOPPER_1.PINCH_VALVE,
                           THRID_STEP_DONE := "DB17000_MAINTENANCE_GLOBAL_VARIABLES".ACTION_DONE.POWDER.UNIT_1.HOPPER_1.TUBE_SECTION_1,
                           FOURTH_STEP_DONE := "DB17000_MAINTENANCE_GLOBAL_VARIABLES".ACTION_DONE.POWDER.UNIT_1.HOPPER_1.TUBE_SECTION_2,
                           FIFTH_STEP_DONE := 0,
                           SIXTH_STEP_DONE := 0,
                           SEVENTH_STEP_DONE := 0,
                           FIRST_OPERATOR_HELP => "DB17100_MAINTENANCE_OPERATOR_HELP".OPERATOR_HELP[7],
                           SECOND_OPERATOR_HELP => "DB17100_MAINTENANCE_OPERATOR_HELP".OPERATOR_HELP[8],
                           THRID_OPERATOR_HELP => "DB17100_MAINTENANCE_OPERATOR_HELP".OPERATOR_HELP[9],
                           FOURTH_OPERATOR_HELP => "DB17100_MAINTENANCE_OPERATOR_HELP".OPERATOR_HELP[10],
                           FIFTH_OPERATOR_HELP => #NULL,
                           SIXTH_OPERATOR_HELP => #NULL,
                           SEVENTH_OPERATOR_HELP => #NULL,
                           MAINTENANCE_IN_PROGRESS => "DB17200_MAINTENANCE_SEQUENCE".MAINTENANCE_IN_PROGRESS[26]);
END_REGION

REGION Network 31: NO FLOW OF POWDER UNIT 1 [1]
   RUNG wire#powerrail
      "FC17900_MAINTENANCE_SEQUENCE"(REQUEST := "DB17200_MAINTENANCE_SEQUENCE".MAINTENANCE_IN_PROGRESS[26], NUMBER_STEPS := 4, FIRST_STEP_DONE := "DB17000_MAINTENANCE_GLOBAL_VARIABLES".ACTION_DONE.POWDER.UNIT_1.HOPPER_2.HOPPER, SECOND_STEP_DONE := "DB17000_MAINTENANCE_GLOBAL_VARIABLES".ACTION_DONE.POWDER.UNIT_1.HOPPER_2.PINCH_VALVE, THRID_STEP_DONE := "DB17000_MAINTENANCE_GLOBAL_VARIABLES".ACTION_DONE.POWDER.UNIT_1.HOPPER_2.TUBE_SECTION_1, FOURTH_STEP_DONE := "DB17000_MAINTENANCE_GLOBAL_VARIABLES".ACTION_DONE.POWDER.UNIT_1.HOPPER_2.TUBE_SECTION_2, FIFTH_STEP_DONE := 0, SIXTH_STEP_DONE := 0, SEVENTH_STEP_DONE := 0, FIRST_OPERATOR_HELP => "DB17100_MAINTENANCE_OPERATOR_HELP".OPERATOR_HELP[12], SECOND_OPERATOR_HELP => "DB17100_MAINTENANCE_OPERATOR_HELP".OPERATOR_HELP[13], THRID_OPERATOR_HELP => "DB17100_MAINTENANCE_OPERATOR_HELP".OPERATOR_HELP[14], FOURTH_OPERATOR_HELP => "DB17100_MAINTENANCE_OPERATOR_HELP".OPERATOR_HELP[15], FIFTH_OPERATOR_HELP => #NULL, SIXTH_OPERATOR_HELP => #NULL, SEVENTH_OPERATOR_HELP => #NULL, MAINTENANCE_IN_PROGRESS => "DB17200_MAINTENANCE_SEQUENCE".MAINTENANCE_IN_PROGRESS[27])
   END_RUNG
   // the same network as SCL:
   "FC17900_MAINTENANCE_SEQUENCE"(REQUEST := "DB17200_MAINTENANCE_SEQUENCE".MAINTENANCE_IN_PROGRESS[26],
                           NUMBER_STEPS := 4,
                           FIRST_STEP_DONE := "DB17000_MAINTENANCE_GLOBAL_VARIABLES".ACTION_DONE.POWDER.UNIT_1.HOPPER_2.HOPPER,
                           SECOND_STEP_DONE := "DB17000_MAINTENANCE_GLOBAL_VARIABLES".ACTION_DONE.POWDER.UNIT_1.HOPPER_2.PINCH_VALVE,
                           THRID_STEP_DONE := "DB17000_MAINTENANCE_GLOBAL_VARIABLES".ACTION_DONE.POWDER.UNIT_1.HOPPER_2.TUBE_SECTION_1,
                           FOURTH_STEP_DONE := "DB17000_MAINTENANCE_GLOBAL_VARIABLES".ACTION_DONE.POWDER.UNIT_1.HOPPER_2.TUBE_SECTION_2,
                           FIFTH_STEP_DONE := 0,
                           SIXTH_STEP_DONE := 0,
                           SEVENTH_STEP_DONE := 0,
                           FIRST_OPERATOR_HELP => "DB17100_MAINTENANCE_OPERATOR_HELP".OPERATOR_HELP[12],
                           SECOND_OPERATOR_HELP => "DB17100_MAINTENANCE_OPERATOR_HELP".OPERATOR_HELP[13],
                           THRID_OPERATOR_HELP => "DB17100_MAINTENANCE_OPERATOR_HELP".OPERATOR_HELP[14],
                           FOURTH_OPERATOR_HELP => "DB17100_MAINTENANCE_OPERATOR_HELP".OPERATOR_HELP[15],
                           FIFTH_OPERATOR_HELP => #NULL,
                           SIXTH_OPERATOR_HELP => #NULL,
                           SEVENTH_OPERATOR_HELP => #NULL,
                           MAINTENANCE_IN_PROGRESS => "DB17200_MAINTENANCE_SEQUENCE".MAINTENANCE_IN_PROGRESS[27]);
END_REGION

REGION Network 32: NO FLOW OF POWDER UNIT 2 [0]
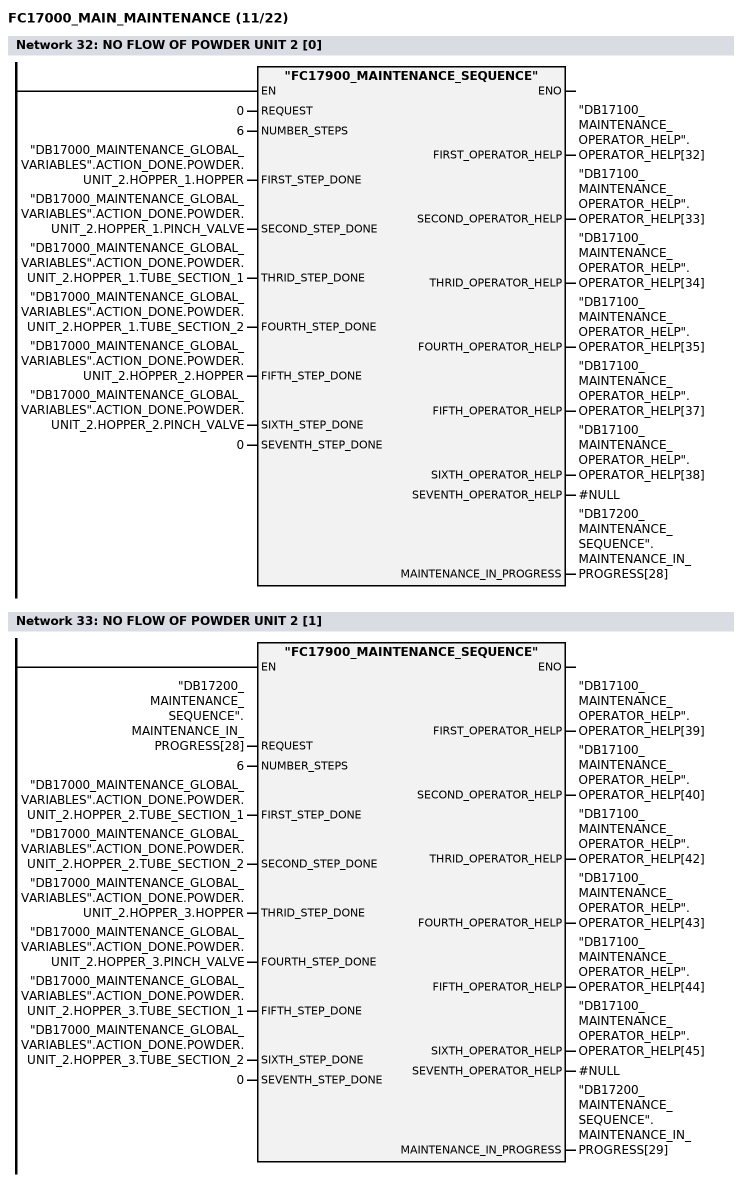
   RUNG wire#powerrail
      "FC17900_MAINTENANCE_SEQUENCE"(REQUEST := 0, NUMBER_STEPS := 6, FIRST_STEP_DONE := "DB17000_MAINTENANCE_GLOBAL_VARIABLES".ACTION_DONE.POWDER.UNIT_2.HOPPER_1.HOPPER, SECOND_STEP_DONE := "DB17000_MAINTENANCE_GLOBAL_VARIABLES".ACTION_DONE.POWDER.UNIT_2.HOPPER_1.PINCH_VALVE, THRID_STEP_DONE := "DB17000_MAINTENANCE_GLOBAL_VARIABLES".ACTION_DONE.POWDER.UNIT_2.HOPPER_1.TUBE_SECTION_1, FOURTH_STEP_DONE := "DB17000_MAINTENANCE_GLOBAL_VARIABLES".ACTION_DONE.POWDER.UNIT_2.HOPPER_1.TUBE_SECTION_2, FIFTH_STEP_DONE := "DB17000_MAINTENANCE_GLOBAL_VARIABLES".ACTION_DONE.POWDER.UNIT_2.HOPPER_2.HOPPER, SIXTH_STEP_DONE := "DB17000_MAINTENANCE_GLOBAL_VARIABLES".ACTION_DONE.POWDER.UNIT_2.HOPPER_2.PINCH_VALVE, SEVENTH_STEP_DONE := 0, FIRST_OPERATOR_HELP => "DB17100_MAINTENANCE_OPERATOR_HELP".OPERATOR_HELP[32], SECOND_OPERATOR_HELP => "DB17100_MAINTENANCE_OPERATOR_HELP".OPERATOR_HELP[33], THRID_OPERATOR_HELP => "DB17100_MAINTENANCE_OPERATOR_HELP".OPERATOR_HELP[34], FOURTH_OPERATOR_HELP => "DB17100_MAINTENANCE_OPERATOR_HELP".OPERATOR_HELP[35], FIFTH_OPERATOR_HELP => "DB17100_MAINTENANCE_OPERATOR_HELP".OPERATOR_HELP[37], SIXTH_OPERATOR_HELP => "DB17100_MAINTENANCE_OPERATOR_HELP".OPERATOR_HELP[38], SEVENTH_OPERATOR_HELP => #NULL, MAINTENANCE_IN_PROGRESS => "DB17200_MAINTENANCE_SEQUENCE".MAINTENANCE_IN_PROGRESS[28])
   END_RUNG
   // the same network as SCL:
   "FC17900_MAINTENANCE_SEQUENCE"(REQUEST := 0,
                           NUMBER_STEPS := 6,
                           FIRST_STEP_DONE := "DB17000_MAINTENANCE_GLOBAL_VARIABLES".ACTION_DONE.POWDER.UNIT_2.HOPPER_1.HOPPER,
                           SECOND_STEP_DONE := "DB17000_MAINTENANCE_GLOBAL_VARIABLES".ACTION_DONE.POWDER.UNIT_2.HOPPER_1.PINCH_VALVE,
                           THRID_STEP_DONE := "DB17000_MAINTENANCE_GLOBAL_VARIABLES".ACTION_DONE.POWDER.UNIT_2.HOPPER_1.TUBE_SECTION_1,
                           FOURTH_STEP_DONE := "DB17000_MAINTENANCE_GLOBAL_VARIABLES".ACTION_DONE.POWDER.UNIT_2.HOPPER_1.TUBE_SECTION_2,
                           FIFTH_STEP_DONE := "DB17000_MAINTENANCE_GLOBAL_VARIABLES".ACTION_DONE.POWDER.UNIT_2.HOPPER_2.HOPPER,
                           SIXTH_STEP_DONE := "DB17000_MAINTENANCE_GLOBAL_VARIABLES".ACTION_DONE.POWDER.UNIT_2.HOPPER_2.PINCH_VALVE,
                           SEVENTH_STEP_DONE := 0,
                           FIRST_OPERATOR_HELP => "DB17100_MAINTENANCE_OPERATOR_HELP".OPERATOR_HELP[32],
                           SECOND_OPERATOR_HELP => "DB17100_MAINTENANCE_OPERATOR_HELP".OPERATOR_HELP[33],
                           THRID_OPERATOR_HELP => "DB17100_MAINTENANCE_OPERATOR_HELP".OPERATOR_HELP[34],
                           FOURTH_OPERATOR_HELP => "DB17100_MAINTENANCE_OPERATOR_HELP".OPERATOR_HELP[35],
                           FIFTH_OPERATOR_HELP => "DB17100_MAINTENANCE_OPERATOR_HELP".OPERATOR_HELP[37],
                           SIXTH_OPERATOR_HELP => "DB17100_MAINTENANCE_OPERATOR_HELP".OPERATOR_HELP[38],
                           SEVENTH_OPERATOR_HELP => #NULL,
                           MAINTENANCE_IN_PROGRESS => "DB17200_MAINTENANCE_SEQUENCE".MAINTENANCE_IN_PROGRESS[28]);
END_REGION

REGION Network 33: NO FLOW OF POWDER UNIT 2 [1]
   RUNG wire#powerrail
      "FC17900_MAINTENANCE_SEQUENCE"(REQUEST := "DB17200_MAINTENANCE_SEQUENCE".MAINTENANCE_IN_PROGRESS[28], NUMBER_STEPS := 6, FIRST_STEP_DONE := "DB17000_MAINTENANCE_GLOBAL_VARIABLES".ACTION_DONE.POWDER.UNIT_2.HOPPER_2.TUBE_SECTION_1, SECOND_STEP_DONE := "DB17000_MAINTENANCE_GLOBAL_VARIABLES".ACTION_DONE.POWDER.UNIT_2.HOPPER_2.TUBE_SECTION_2, THRID_STEP_DONE := "DB17000_MAINTENANCE_GLOBAL_VARIABLES".ACTION_DONE.POWDER.UNIT_2.HOPPER_3.HOPPER, FOURTH_STEP_DONE := "DB17000_MAINTENANCE_GLOBAL_VARIABLES".ACTION_DONE.POWDER.UNIT_2.HOPPER_3.PINCH_VALVE, FIFTH_STEP_DONE := "DB17000_MAINTENANCE_GLOBAL_VARIABLES".ACTION_DONE.POWDER.UNIT_2.HOPPER_3.TUBE_SECTION_1, SIXTH_STEP_DONE := "DB17000_MAINTENANCE_GLOBAL_VARIABLES".ACTION_DONE.POWDER.UNIT_2.HOPPER_3.TUBE_SECTION_2, SEVENTH_STEP_DONE := 0, FIRST_OPERATOR_HELP => "DB17100_MAINTENANCE_OPERATOR_HELP".OPERATOR_HELP[39], SECOND_OPERATOR_HELP => "DB17100_MAINTENANCE_OPERATOR_HELP".OPERATOR_HELP[40], THRID_OPERATOR_HELP => "DB17100_MAINTENANCE_OPERATOR_HELP".OPERATOR_HELP[42], FOURTH_OPERATOR_HELP => "DB17100_MAINTENANCE_OPERATOR_HELP".OPERATOR_HELP[43], FIFTH_OPERATOR_HELP => "DB17100_MAINTENANCE_OPERATOR_HELP".OPERATOR_HELP[44], SIXTH_OPERATOR_HELP => "DB17100_MAINTENANCE_OPERATOR_HELP".OPERATOR_HELP[45], SEVENTH_OPERATOR_HELP => #NULL, MAINTENANCE_IN_PROGRESS => "DB17200_MAINTENANCE_SEQUENCE".MAINTENANCE_IN_PROGRESS[29])
   END_RUNG
   // the same network as SCL:
   "FC17900_MAINTENANCE_SEQUENCE"(REQUEST := "DB17200_MAINTENANCE_SEQUENCE".MAINTENANCE_IN_PROGRESS[28],
                           NUMBER_STEPS := 6,
                           FIRST_STEP_DONE := "DB17000_MAINTENANCE_GLOBAL_VARIABLES".ACTION_DONE.POWDER.UNIT_2.HOPPER_2.TUBE_SECTION_1,
                           SECOND_STEP_DONE := "DB17000_MAINTENANCE_GLOBAL_VARIABLES".ACTION_DONE.POWDER.UNIT_2.HOPPER_2.TUBE_SECTION_2,
                           THRID_STEP_DONE := "DB17000_MAINTENANCE_GLOBAL_VARIABLES".ACTION_DONE.POWDER.UNIT_2.HOPPER_3.HOPPER,
                           FOURTH_STEP_DONE := "DB17000_MAINTENANCE_GLOBAL_VARIABLES".ACTION_DONE.POWDER.UNIT_2.HOPPER_3.PINCH_VALVE,
                           FIFTH_STEP_DONE := "DB17000_MAINTENANCE_GLOBAL_VARIABLES".ACTION_DONE.POWDER.UNIT_2.HOPPER_3.TUBE_SECTION_1,
                           SIXTH_STEP_DONE := "DB17000_MAINTENANCE_GLOBAL_VARIABLES".ACTION_DONE.POWDER.UNIT_2.HOPPER_3.TUBE_SECTION_2,
                           SEVENTH_STEP_DONE := 0,
                           FIRST_OPERATOR_HELP => "DB17100_MAINTENANCE_OPERATOR_HELP".OPERATOR_HELP[39],
                           SECOND_OPERATOR_HELP => "DB17100_MAINTENANCE_OPERATOR_HELP".OPERATOR_HELP[40],
                           THRID_OPERATOR_HELP => "DB17100_MAINTENANCE_OPERATOR_HELP".OPERATOR_HELP[42],
                           FOURTH_OPERATOR_HELP => "DB17100_MAINTENANCE_OPERATOR_HELP".OPERATOR_HELP[43],
                           FIFTH_OPERATOR_HELP => "DB17100_MAINTENANCE_OPERATOR_HELP".OPERATOR_HELP[44],
                           SIXTH_OPERATOR_HELP => "DB17100_MAINTENANCE_OPERATOR_HELP".OPERATOR_HELP[45],
                           SEVENTH_OPERATOR_HELP => #NULL,
                           MAINTENANCE_IN_PROGRESS => "DB17200_MAINTENANCE_SEQUENCE".MAINTENANCE_IN_PROGRESS[29]);
END_REGION

REGION Network 34: WRONG GR/MIN UNIT 1
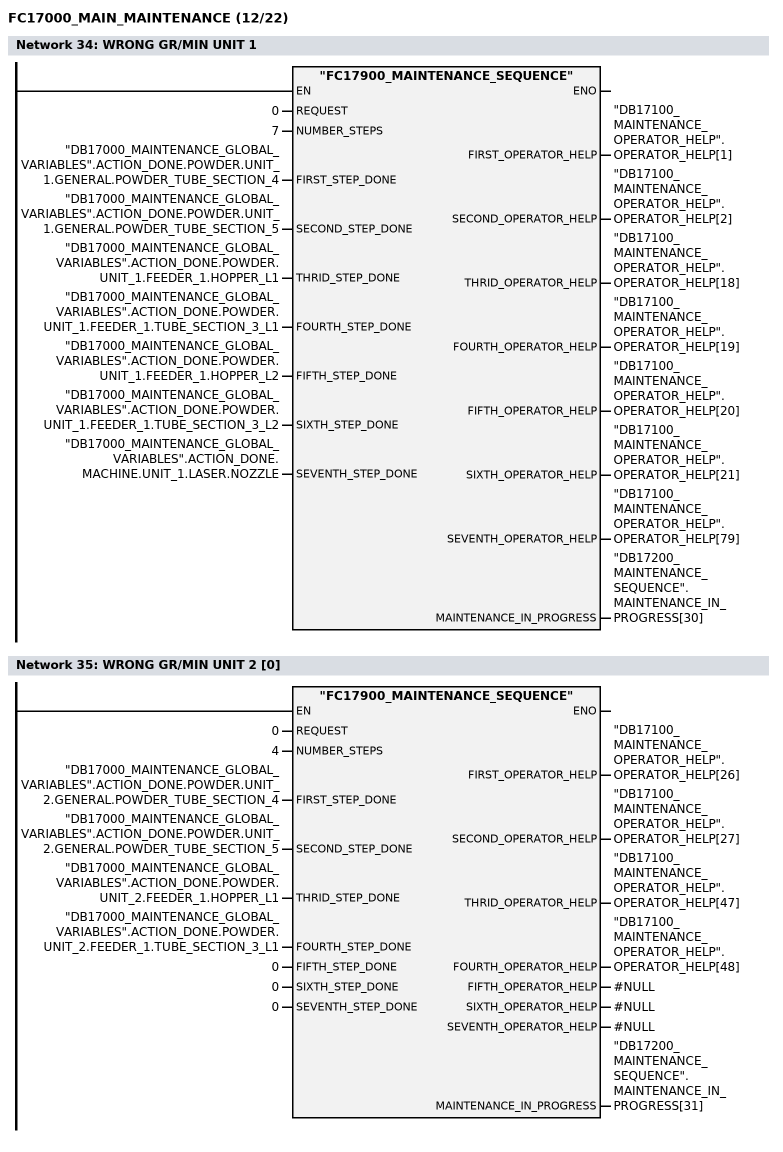
   RUNG wire#powerrail
      "FC17900_MAINTENANCE_SEQUENCE"(REQUEST := 0, NUMBER_STEPS := 7, FIRST_STEP_DONE := "DB17000_MAINTENANCE_GLOBAL_VARIABLES".ACTION_DONE.POWDER.UNIT_1.GENERAL.POWDER_TUBE_SECTION_4, SECOND_STEP_DONE := "DB17000_MAINTENANCE_GLOBAL_VARIABLES".ACTION_DONE.POWDER.UNIT_1.GENERAL.POWDER_TUBE_SECTION_5, THRID_STEP_DONE := "DB17000_MAINTENANCE_GLOBAL_VARIABLES".ACTION_DONE.POWDER.UNIT_1.FEEDER_1.HOPPER_L1, FOURTH_STEP_DONE := "DB17000_MAINTENANCE_GLOBAL_VARIABLES".ACTION_DONE.POWDER.UNIT_1.FEEDER_1.TUBE_SECTION_3_L1, FIFTH_STEP_DONE := "DB17000_MAINTENANCE_GLOBAL_VARIABLES".ACTION_DONE.POWDER.UNIT_1.FEEDER_1.HOPPER_L2, SIXTH_STEP_DONE := "DB17000_MAINTENANCE_GLOBAL_VARIABLES".ACTION_DONE.POWDER.UNIT_1.FEEDER_1.TUBE_SECTION_3_L2, SEVENTH_STEP_DONE := "DB17000_MAINTENANCE_GLOBAL_VARIABLES".ACTION_DONE.MACHINE.UNIT_1.LASER.NOZZLE, FIRST_OPERATOR_HELP => "DB17100_MAINTENANCE_OPERATOR_HELP".OPERATOR_HELP[1], SECOND_OPERATOR_HELP => "DB17100_MAINTENANCE_OPERATOR_HELP".OPERATOR_HELP[2], THRID_OPERATOR_HELP => "DB17100_MAINTENANCE_OPERATOR_HELP".OPERATOR_HELP[18], FOURTH_OPERATOR_HELP => "DB17100_MAINTENANCE_OPERATOR_HELP".OPERATOR_HELP[19], FIFTH_OPERATOR_HELP => "DB17100_MAINTENANCE_OPERATOR_HELP".OPERATOR_HELP[20], SIXTH_OPERATOR_HELP => "DB17100_MAINTENANCE_OPERATOR_HELP".OPERATOR_HELP[21], SEVENTH_OPERATOR_HELP => "DB17100_MAINTENANCE_OPERATOR_HELP".OPERATOR_HELP[79], MAINTENANCE_IN_PROGRESS => "DB17200_MAINTENANCE_SEQUENCE".MAINTENANCE_IN_PROGRESS[30])
   END_RUNG
   // the same network as SCL:
   "FC17900_MAINTENANCE_SEQUENCE"(REQUEST := 0,
                           NUMBER_STEPS := 7,
                           FIRST_STEP_DONE := "DB17000_MAINTENANCE_GLOBAL_VARIABLES".ACTION_DONE.POWDER.UNIT_1.GENERAL.POWDER_TUBE_SECTION_4,
                           SECOND_STEP_DONE := "DB17000_MAINTENANCE_GLOBAL_VARIABLES".ACTION_DONE.POWDER.UNIT_1.GENERAL.POWDER_TUBE_SECTION_5,
                           THRID_STEP_DONE := "DB17000_MAINTENANCE_GLOBAL_VARIABLES".ACTION_DONE.POWDER.UNIT_1.FEEDER_1.HOPPER_L1,
                           FOURTH_STEP_DONE := "DB17000_MAINTENANCE_GLOBAL_VARIABLES".ACTION_DONE.POWDER.UNIT_1.FEEDER_1.TUBE_SECTION_3_L1,
                           FIFTH_STEP_DONE := "DB17000_MAINTENANCE_GLOBAL_VARIABLES".ACTION_DONE.POWDER.UNIT_1.FEEDER_1.HOPPER_L2,
                           SIXTH_STEP_DONE := "DB17000_MAINTENANCE_GLOBAL_VARIABLES".ACTION_DONE.POWDER.UNIT_1.FEEDER_1.TUBE_SECTION_3_L2,
                           SEVENTH_STEP_DONE := "DB17000_MAINTENANCE_GLOBAL_VARIABLES".ACTION_DONE.MACHINE.UNIT_1.LASER.NOZZLE,
                           FIRST_OPERATOR_HELP => "DB17100_MAINTENANCE_OPERATOR_HELP".OPERATOR_HELP[1],
                           SECOND_OPERATOR_HELP => "DB17100_MAINTENANCE_OPERATOR_HELP".OPERATOR_HELP[2],
                           THRID_OPERATOR_HELP => "DB17100_MAINTENANCE_OPERATOR_HELP".OPERATOR_HELP[18],
                           FOURTH_OPERATOR_HELP => "DB17100_MAINTENANCE_OPERATOR_HELP".OPERATOR_HELP[19],
                           FIFTH_OPERATOR_HELP => "DB17100_MAINTENANCE_OPERATOR_HELP".OPERATOR_HELP[20],
                           SIXTH_OPERATOR_HELP => "DB17100_MAINTENANCE_OPERATOR_HELP".OPERATOR_HELP[21],
                           SEVENTH_OPERATOR_HELP => "DB17100_MAINTENANCE_OPERATOR_HELP".OPERATOR_HELP[79],
                           MAINTENANCE_IN_PROGRESS => "DB17200_MAINTENANCE_SEQUENCE".MAINTENANCE_IN_PROGRESS[30]);
END_REGION

REGION Network 35: WRONG GR/MIN UNIT 2 [0]
   RUNG wire#powerrail
      "FC17900_MAINTENANCE_SEQUENCE"(REQUEST := 0, NUMBER_STEPS := 4, FIRST_STEP_DONE := "DB17000_MAINTENANCE_GLOBAL_VARIABLES".ACTION_DONE.POWDER.UNIT_2.GENERAL.POWDER_TUBE_SECTION_4, SECOND_STEP_DONE := "DB17000_MAINTENANCE_GLOBAL_VARIABLES".ACTION_DONE.POWDER.UNIT_2.GENERAL.POWDER_TUBE_SECTION_5, THRID_STEP_DONE := "DB17000_MAINTENANCE_GLOBAL_VARIABLES".ACTION_DONE.POWDER.UNIT_2.FEEDER_1.HOPPER_L1, FOURTH_STEP_DONE := "DB17000_MAINTENANCE_GLOBAL_VARIABLES".ACTION_DONE.POWDER.UNIT_2.FEEDER_1.TUBE_SECTION_3_L1, FIFTH_STEP_DONE := 0, SIXTH_STEP_DONE := 0, SEVENTH_STEP_DONE := 0, FIRST_OPERATOR_HELP => "DB17100_MAINTENANCE_OPERATOR_HELP".OPERATOR_HELP[26], SECOND_OPERATOR_HELP => "DB17100_MAINTENANCE_OPERATOR_HELP".OPERATOR_HELP[27], THRID_OPERATOR_HELP => "DB17100_MAINTENANCE_OPERATOR_HELP".OPERATOR_HELP[47], FOURTH_OPERATOR_HELP => "DB17100_MAINTENANCE_OPERATOR_HELP".OPERATOR_HELP[48], FIFTH_OPERATOR_HELP => #NULL, SIXTH_OPERATOR_HELP => #NULL, SEVENTH_OPERATOR_HELP => #NULL, MAINTENANCE_IN_PROGRESS => "DB17200_MAINTENANCE_SEQUENCE".MAINTENANCE_IN_PROGRESS[31])
   END_RUNG
   // the same network as SCL:
   "FC17900_MAINTENANCE_SEQUENCE"(REQUEST := 0,
                           NUMBER_STEPS := 4,
                           FIRST_STEP_DONE := "DB17000_MAINTENANCE_GLOBAL_VARIABLES".ACTION_DONE.POWDER.UNIT_2.GENERAL.POWDER_TUBE_SECTION_4,
                           SECOND_STEP_DONE := "DB17000_MAINTENANCE_GLOBAL_VARIABLES".ACTION_DONE.POWDER.UNIT_2.GENERAL.POWDER_TUBE_SECTION_5,
                           THRID_STEP_DONE := "DB17000_MAINTENANCE_GLOBAL_VARIABLES".ACTION_DONE.POWDER.UNIT_2.FEEDER_1.HOPPER_L1,
                           FOURTH_STEP_DONE := "DB17000_MAINTENANCE_GLOBAL_VARIABLES".ACTION_DONE.POWDER.UNIT_2.FEEDER_1.TUBE_SECTION_3_L1,
                           FIFTH_STEP_DONE := 0,
                           SIXTH_STEP_DONE := 0,
                           SEVENTH_STEP_DONE := 0,
                           FIRST_OPERATOR_HELP => "DB17100_MAINTENANCE_OPERATOR_HELP".OPERATOR_HELP[26],
                           SECOND_OPERATOR_HELP => "DB17100_MAINTENANCE_OPERATOR_HELP".OPERATOR_HELP[27],
                           THRID_OPERATOR_HELP => "DB17100_MAINTENANCE_OPERATOR_HELP".OPERATOR_HELP[47],
                           FOURTH_OPERATOR_HELP => "DB17100_MAINTENANCE_OPERATOR_HELP".OPERATOR_HELP[48],
                           FIFTH_OPERATOR_HELP => #NULL,
                           SIXTH_OPERATOR_HELP => #NULL,
                           SEVENTH_OPERATOR_HELP => #NULL,
                           MAINTENANCE_IN_PROGRESS => "DB17200_MAINTENANCE_SEQUENCE".MAINTENANCE_IN_PROGRESS[31]);
END_REGION

REGION Network 36: WRONG GR/MIN UNIT 2 [1]
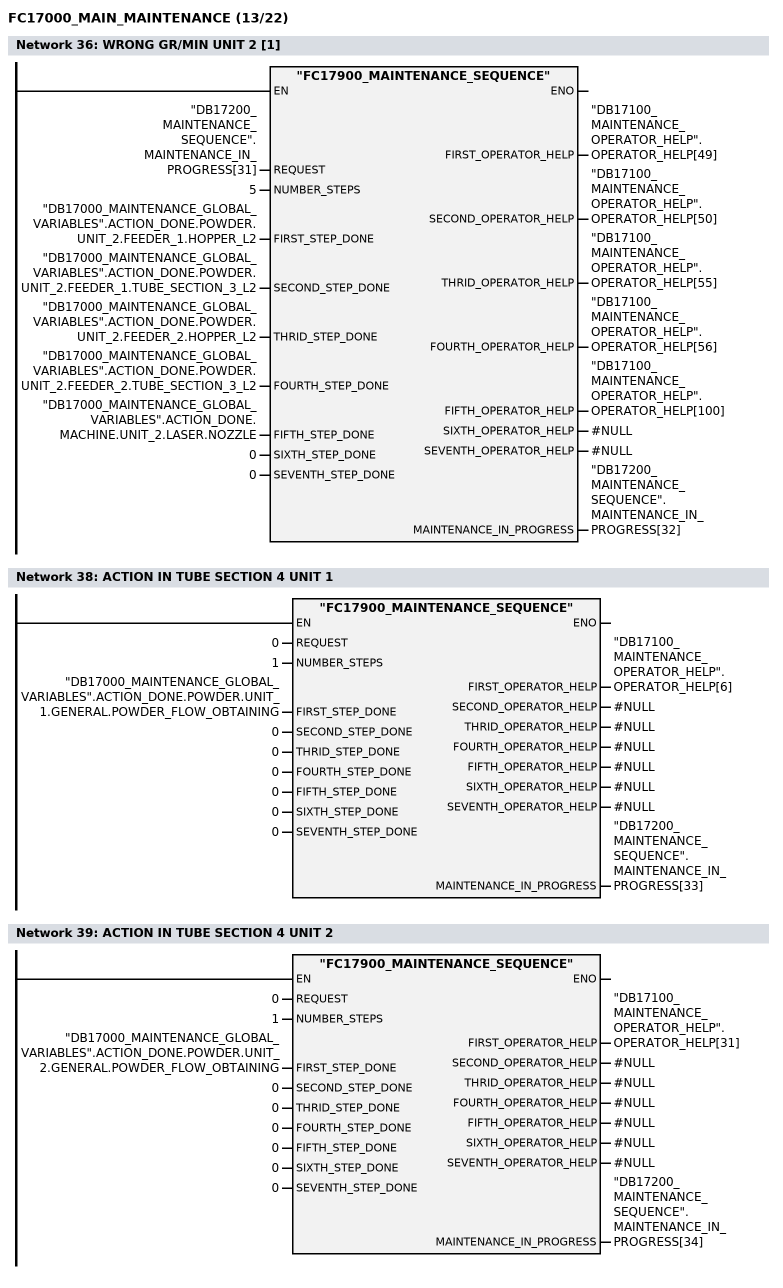
   RUNG wire#powerrail
      "FC17900_MAINTENANCE_SEQUENCE"(REQUEST := "DB17200_MAINTENANCE_SEQUENCE".MAINTENANCE_IN_PROGRESS[31], NUMBER_STEPS := 5, FIRST_STEP_DONE := "DB17000_MAINTENANCE_GLOBAL_VARIABLES".ACTION_DONE.POWDER.UNIT_2.FEEDER_1.HOPPER_L2, SECOND_STEP_DONE := "DB17000_MAINTENANCE_GLOBAL_VARIABLES".ACTION_DONE.POWDER.UNIT_2.FEEDER_1.TUBE_SECTION_3_L2, THRID_STEP_DONE := "DB17000_MAINTENANCE_GLOBAL_VARIABLES".ACTION_DONE.POWDER.UNIT_2.FEEDER_2.HOPPER_L2, FOURTH_STEP_DONE := "DB17000_MAINTENANCE_GLOBAL_VARIABLES".ACTION_DONE.POWDER.UNIT_2.FEEDER_2.TUBE_SECTION_3_L2, FIFTH_STEP_DONE := "DB17000_MAINTENANCE_GLOBAL_VARIABLES".ACTION_DONE.MACHINE.UNIT_2.LASER.NOZZLE, SIXTH_STEP_DONE := 0, SEVENTH_STEP_DONE := 0, FIRST_OPERATOR_HELP => "DB17100_MAINTENANCE_OPERATOR_HELP".OPERATOR_HELP[49], SECOND_OPERATOR_HELP => "DB17100_MAINTENANCE_OPERATOR_HELP".OPERATOR_HELP[50], THRID_OPERATOR_HELP => "DB17100_MAINTENANCE_OPERATOR_HELP".OPERATOR_HELP[55], FOURTH_OPERATOR_HELP => "DB17100_MAINTENANCE_OPERATOR_HELP".OPERATOR_HELP[56], FIFTH_OPERATOR_HELP => "DB17100_MAINTENANCE_OPERATOR_HELP".OPERATOR_HELP[100], SIXTH_OPERATOR_HELP => #NULL, SEVENTH_OPERATOR_HELP => #NULL, MAINTENANCE_IN_PROGRESS => "DB17200_MAINTENANCE_SEQUENCE".MAINTENANCE_IN_PROGRESS[32])
   END_RUNG
   // the same network as SCL:
   "FC17900_MAINTENANCE_SEQUENCE"(REQUEST := "DB17200_MAINTENANCE_SEQUENCE".MAINTENANCE_IN_PROGRESS[31],
                           NUMBER_STEPS := 5,
                           FIRST_STEP_DONE := "DB17000_MAINTENANCE_GLOBAL_VARIABLES".ACTION_DONE.POWDER.UNIT_2.FEEDER_1.HOPPER_L2,
                           SECOND_STEP_DONE := "DB17000_MAINTENANCE_GLOBAL_VARIABLES".ACTION_DONE.POWDER.UNIT_2.FEEDER_1.TUBE_SECTION_3_L2,
                           THRID_STEP_DONE := "DB17000_MAINTENANCE_GLOBAL_VARIABLES".ACTION_DONE.POWDER.UNIT_2.FEEDER_2.HOPPER_L2,
                           FOURTH_STEP_DONE := "DB17000_MAINTENANCE_GLOBAL_VARIABLES".ACTION_DONE.POWDER.UNIT_2.FEEDER_2.TUBE_SECTION_3_L2,
                           FIFTH_STEP_DONE := "DB17000_MAINTENANCE_GLOBAL_VARIABLES".ACTION_DONE.MACHINE.UNIT_2.LASER.NOZZLE,
                           SIXTH_STEP_DONE := 0,
                           SEVENTH_STEP_DONE := 0,
                           FIRST_OPERATOR_HELP => "DB17100_MAINTENANCE_OPERATOR_HELP".OPERATOR_HELP[49],
                           SECOND_OPERATOR_HELP => "DB17100_MAINTENANCE_OPERATOR_HELP".OPERATOR_HELP[50],
                           THRID_OPERATOR_HELP => "DB17100_MAINTENANCE_OPERATOR_HELP".OPERATOR_HELP[55],
                           FOURTH_OPERATOR_HELP => "DB17100_MAINTENANCE_OPERATOR_HELP".OPERATOR_HELP[56],
                           FIFTH_OPERATOR_HELP => "DB17100_MAINTENANCE_OPERATOR_HELP".OPERATOR_HELP[100],
                           SIXTH_OPERATOR_HELP => #NULL,
                           SEVENTH_OPERATOR_HELP => #NULL,
                           MAINTENANCE_IN_PROGRESS => "DB17200_MAINTENANCE_SEQUENCE".MAINTENANCE_IN_PROGRESS[32]);
END_REGION

REGION Network 37: <<<---MAINTENANCE EVENTS--->>>
END_REGION

REGION Network 38: ACTION IN TUBE SECTION 4 UNIT 1
   RUNG wire#powerrail
      "FC17900_MAINTENANCE_SEQUENCE"(REQUEST := 0, NUMBER_STEPS := 1, FIRST_STEP_DONE := "DB17000_MAINTENANCE_GLOBAL_VARIABLES".ACTION_DONE.POWDER.UNIT_1.GENERAL.POWDER_FLOW_OBTAINING, SECOND_STEP_DONE := 0, THRID_STEP_DONE := 0, FOURTH_STEP_DONE := 0, FIFTH_STEP_DONE := 0, SIXTH_STEP_DONE := 0, SEVENTH_STEP_DONE := 0, FIRST_OPERATOR_HELP => "DB17100_MAINTENANCE_OPERATOR_HELP".OPERATOR_HELP[6], SECOND_OPERATOR_HELP => #NULL, THRID_OPERATOR_HELP => #NULL, FOURTH_OPERATOR_HELP => #NULL, FIFTH_OPERATOR_HELP => #NULL, SIXTH_OPERATOR_HELP => #NULL, SEVENTH_OPERATOR_HELP => #NULL, MAINTENANCE_IN_PROGRESS => "DB17200_MAINTENANCE_SEQUENCE".MAINTENANCE_IN_PROGRESS[33])
   END_RUNG
   // the same network as SCL:
   "FC17900_MAINTENANCE_SEQUENCE"(REQUEST := 0,
                           NUMBER_STEPS := 1,
                           FIRST_STEP_DONE := "DB17000_MAINTENANCE_GLOBAL_VARIABLES".ACTION_DONE.POWDER.UNIT_1.GENERAL.POWDER_FLOW_OBTAINING,
                           SECOND_STEP_DONE := 0,
                           THRID_STEP_DONE := 0,
                           FOURTH_STEP_DONE := 0,
                           FIFTH_STEP_DONE := 0,
                           SIXTH_STEP_DONE := 0,
                           SEVENTH_STEP_DONE := 0,
                           FIRST_OPERATOR_HELP => "DB17100_MAINTENANCE_OPERATOR_HELP".OPERATOR_HELP[6],
                           SECOND_OPERATOR_HELP => #NULL,
                           THRID_OPERATOR_HELP => #NULL,
                           FOURTH_OPERATOR_HELP => #NULL,
                           FIFTH_OPERATOR_HELP => #NULL,
                           SIXTH_OPERATOR_HELP => #NULL,
                           SEVENTH_OPERATOR_HELP => #NULL,
                           MAINTENANCE_IN_PROGRESS => "DB17200_MAINTENANCE_SEQUENCE".MAINTENANCE_IN_PROGRESS[33]);
END_REGION

REGION Network 39: ACTION IN TUBE SECTION 4 UNIT 2
   RUNG wire#powerrail
      "FC17900_MAINTENANCE_SEQUENCE"(REQUEST := 0, NUMBER_STEPS := 1, FIRST_STEP_DONE := "DB17000_MAINTENANCE_GLOBAL_VARIABLES".ACTION_DONE.POWDER.UNIT_2.GENERAL.POWDER_FLOW_OBTAINING, SECOND_STEP_DONE := 0, THRID_STEP_DONE := 0, FOURTH_STEP_DONE := 0, FIFTH_STEP_DONE := 0, SIXTH_STEP_DONE := 0, SEVENTH_STEP_DONE := 0, FIRST_OPERATOR_HELP => "DB17100_MAINTENANCE_OPERATOR_HELP".OPERATOR_HELP[31], SECOND_OPERATOR_HELP => #NULL, THRID_OPERATOR_HELP => #NULL, FOURTH_OPERATOR_HELP => #NULL, FIFTH_OPERATOR_HELP => #NULL, SIXTH_OPERATOR_HELP => #NULL, SEVENTH_OPERATOR_HELP => #NULL, MAINTENANCE_IN_PROGRESS => "DB17200_MAINTENANCE_SEQUENCE".MAINTENANCE_IN_PROGRESS[34])
   END_RUNG
   // the same network as SCL:
   "FC17900_MAINTENANCE_SEQUENCE"(REQUEST := 0,
                           NUMBER_STEPS := 1,
                           FIRST_STEP_DONE := "DB17000_MAINTENANCE_GLOBAL_VARIABLES".ACTION_DONE.POWDER.UNIT_2.GENERAL.POWDER_FLOW_OBTAINING,
                           SECOND_STEP_DONE := 0,
                           THRID_STEP_DONE := 0,
                           FOURTH_STEP_DONE := 0,
                           FIFTH_STEP_DONE := 0,
                           SIXTH_STEP_DONE := 0,
                           SEVENTH_STEP_DONE := 0,
                           FIRST_OPERATOR_HELP => "DB17100_MAINTENANCE_OPERATOR_HELP".OPERATOR_HELP[31],
                           SECOND_OPERATOR_HELP => #NULL,
                           THRID_OPERATOR_HELP => #NULL,
                           FOURTH_OPERATOR_HELP => #NULL,
                           FIFTH_OPERATOR_HELP => #NULL,
                           SIXTH_OPERATOR_HELP => #NULL,
                           SEVENTH_OPERATOR_HELP => #NULL,
                           MAINTENANCE_IN_PROGRESS => "DB17200_MAINTENANCE_SEQUENCE".MAINTENANCE_IN_PROGRESS[34]);
END_REGION

REGION Network 40: ACTION IN TUBE SECTION 5 UNIT 1
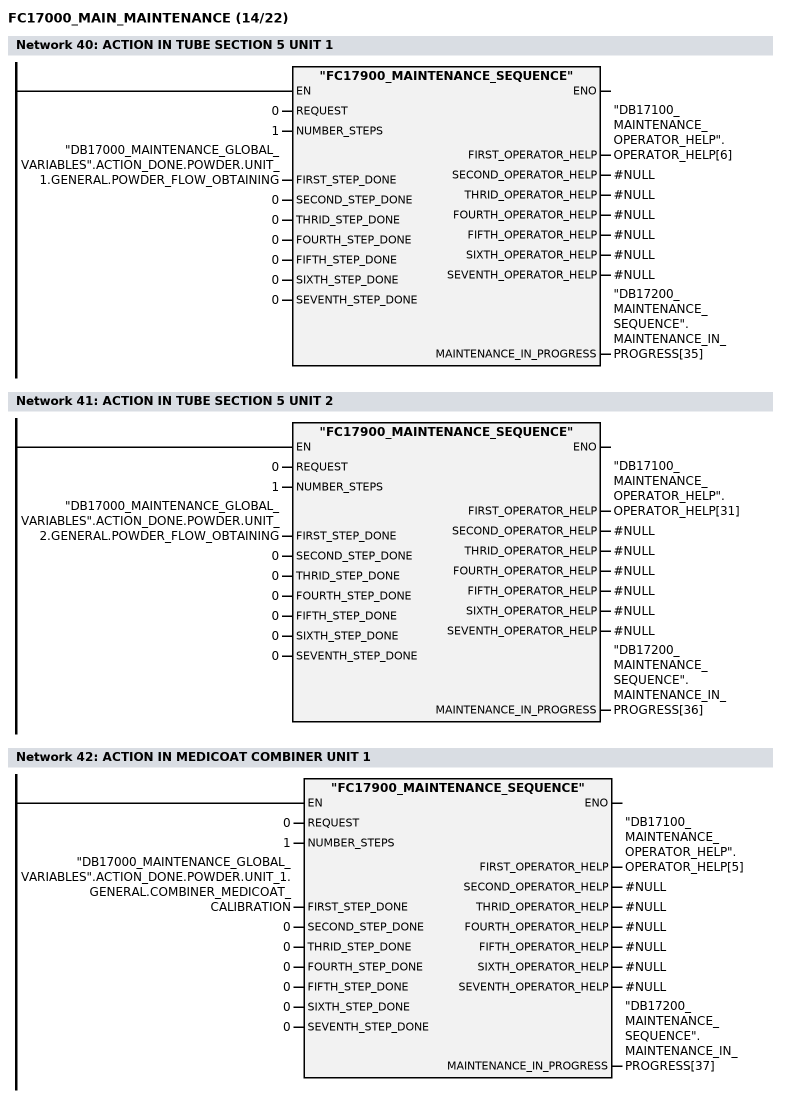
   RUNG wire#powerrail
      "FC17900_MAINTENANCE_SEQUENCE"(REQUEST := 0, NUMBER_STEPS := 1, FIRST_STEP_DONE := "DB17000_MAINTENANCE_GLOBAL_VARIABLES".ACTION_DONE.POWDER.UNIT_1.GENERAL.POWDER_FLOW_OBTAINING, SECOND_STEP_DONE := 0, THRID_STEP_DONE := 0, FOURTH_STEP_DONE := 0, FIFTH_STEP_DONE := 0, SIXTH_STEP_DONE := 0, SEVENTH_STEP_DONE := 0, FIRST_OPERATOR_HELP => "DB17100_MAINTENANCE_OPERATOR_HELP".OPERATOR_HELP[6], SECOND_OPERATOR_HELP => #NULL, THRID_OPERATOR_HELP => #NULL, FOURTH_OPERATOR_HELP => #NULL, FIFTH_OPERATOR_HELP => #NULL, SIXTH_OPERATOR_HELP => #NULL, SEVENTH_OPERATOR_HELP => #NULL, MAINTENANCE_IN_PROGRESS => "DB17200_MAINTENANCE_SEQUENCE".MAINTENANCE_IN_PROGRESS[35])
   END_RUNG
   // the same network as SCL:
   "FC17900_MAINTENANCE_SEQUENCE"(REQUEST := 0,
                           NUMBER_STEPS := 1,
                           FIRST_STEP_DONE := "DB17000_MAINTENANCE_GLOBAL_VARIABLES".ACTION_DONE.POWDER.UNIT_1.GENERAL.POWDER_FLOW_OBTAINING,
                           SECOND_STEP_DONE := 0,
                           THRID_STEP_DONE := 0,
                           FOURTH_STEP_DONE := 0,
                           FIFTH_STEP_DONE := 0,
                           SIXTH_STEP_DONE := 0,
                           SEVENTH_STEP_DONE := 0,
                           FIRST_OPERATOR_HELP => "DB17100_MAINTENANCE_OPERATOR_HELP".OPERATOR_HELP[6],
                           SECOND_OPERATOR_HELP => #NULL,
                           THRID_OPERATOR_HELP => #NULL,
                           FOURTH_OPERATOR_HELP => #NULL,
                           FIFTH_OPERATOR_HELP => #NULL,
                           SIXTH_OPERATOR_HELP => #NULL,
                           SEVENTH_OPERATOR_HELP => #NULL,
                           MAINTENANCE_IN_PROGRESS => "DB17200_MAINTENANCE_SEQUENCE".MAINTENANCE_IN_PROGRESS[35]);
END_REGION

REGION Network 41: ACTION IN TUBE SECTION 5 UNIT 2
   RUNG wire#powerrail
      "FC17900_MAINTENANCE_SEQUENCE"(REQUEST := 0, NUMBER_STEPS := 1, FIRST_STEP_DONE := "DB17000_MAINTENANCE_GLOBAL_VARIABLES".ACTION_DONE.POWDER.UNIT_2.GENERAL.POWDER_FLOW_OBTAINING, SECOND_STEP_DONE := 0, THRID_STEP_DONE := 0, FOURTH_STEP_DONE := 0, FIFTH_STEP_DONE := 0, SIXTH_STEP_DONE := 0, SEVENTH_STEP_DONE := 0, FIRST_OPERATOR_HELP => "DB17100_MAINTENANCE_OPERATOR_HELP".OPERATOR_HELP[31], SECOND_OPERATOR_HELP => #NULL, THRID_OPERATOR_HELP => #NULL, FOURTH_OPERATOR_HELP => #NULL, FIFTH_OPERATOR_HELP => #NULL, SIXTH_OPERATOR_HELP => #NULL, SEVENTH_OPERATOR_HELP => #NULL, MAINTENANCE_IN_PROGRESS => "DB17200_MAINTENANCE_SEQUENCE".MAINTENANCE_IN_PROGRESS[36])
   END_RUNG
   // the same network as SCL:
   "FC17900_MAINTENANCE_SEQUENCE"(REQUEST := 0,
                           NUMBER_STEPS := 1,
                           FIRST_STEP_DONE := "DB17000_MAINTENANCE_GLOBAL_VARIABLES".ACTION_DONE.POWDER.UNIT_2.GENERAL.POWDER_FLOW_OBTAINING,
                           SECOND_STEP_DONE := 0,
                           THRID_STEP_DONE := 0,
                           FOURTH_STEP_DONE := 0,
                           FIFTH_STEP_DONE := 0,
                           SIXTH_STEP_DONE := 0,
                           SEVENTH_STEP_DONE := 0,
                           FIRST_OPERATOR_HELP => "DB17100_MAINTENANCE_OPERATOR_HELP".OPERATOR_HELP[31],
                           SECOND_OPERATOR_HELP => #NULL,
                           THRID_OPERATOR_HELP => #NULL,
                           FOURTH_OPERATOR_HELP => #NULL,
                           FIFTH_OPERATOR_HELP => #NULL,
                           SIXTH_OPERATOR_HELP => #NULL,
                           SEVENTH_OPERATOR_HELP => #NULL,
                           MAINTENANCE_IN_PROGRESS => "DB17200_MAINTENANCE_SEQUENCE".MAINTENANCE_IN_PROGRESS[36]);
END_REGION

REGION Network 42: ACTION IN MEDICOAT COMBINER UNIT 1
   RUNG wire#powerrail
      "FC17900_MAINTENANCE_SEQUENCE"(REQUEST := 0, NUMBER_STEPS := 1, FIRST_STEP_DONE := "DB17000_MAINTENANCE_GLOBAL_VARIABLES".ACTION_DONE.POWDER.UNIT_1.GENERAL.COMBINER_MEDICOAT_CALIBRATION, SECOND_STEP_DONE := 0, THRID_STEP_DONE := 0, FOURTH_STEP_DONE := 0, FIFTH_STEP_DONE := 0, SIXTH_STEP_DONE := 0, SEVENTH_STEP_DONE := 0, FIRST_OPERATOR_HELP => "DB17100_MAINTENANCE_OPERATOR_HELP".OPERATOR_HELP[5], SECOND_OPERATOR_HELP => #NULL, THRID_OPERATOR_HELP => #NULL, FOURTH_OPERATOR_HELP => #NULL, FIFTH_OPERATOR_HELP => #NULL, SIXTH_OPERATOR_HELP => #NULL, SEVENTH_OPERATOR_HELP => #NULL, MAINTENANCE_IN_PROGRESS => "DB17200_MAINTENANCE_SEQUENCE".MAINTENANCE_IN_PROGRESS[37])
   END_RUNG
   // the same network as SCL:
   "FC17900_MAINTENANCE_SEQUENCE"(REQUEST := 0,
                           NUMBER_STEPS := 1,
                           FIRST_STEP_DONE := "DB17000_MAINTENANCE_GLOBAL_VARIABLES".ACTION_DONE.POWDER.UNIT_1.GENERAL.COMBINER_MEDICOAT_CALIBRATION,
                           SECOND_STEP_DONE := 0,
                           THRID_STEP_DONE := 0,
                           FOURTH_STEP_DONE := 0,
                           FIFTH_STEP_DONE := 0,
                           SIXTH_STEP_DONE := 0,
                           SEVENTH_STEP_DONE := 0,
                           FIRST_OPERATOR_HELP => "DB17100_MAINTENANCE_OPERATOR_HELP".OPERATOR_HELP[5],
                           SECOND_OPERATOR_HELP => #NULL,
                           THRID_OPERATOR_HELP => #NULL,
                           FOURTH_OPERATOR_HELP => #NULL,
                           FIFTH_OPERATOR_HELP => #NULL,
                           SIXTH_OPERATOR_HELP => #NULL,
                           SEVENTH_OPERATOR_HELP => #NULL,
                           MAINTENANCE_IN_PROGRESS => "DB17200_MAINTENANCE_SEQUENCE".MAINTENANCE_IN_PROGRESS[37]);
END_REGION

REGION Network 43: ACTION IN MEDICOAT COMBINER UNIT 2
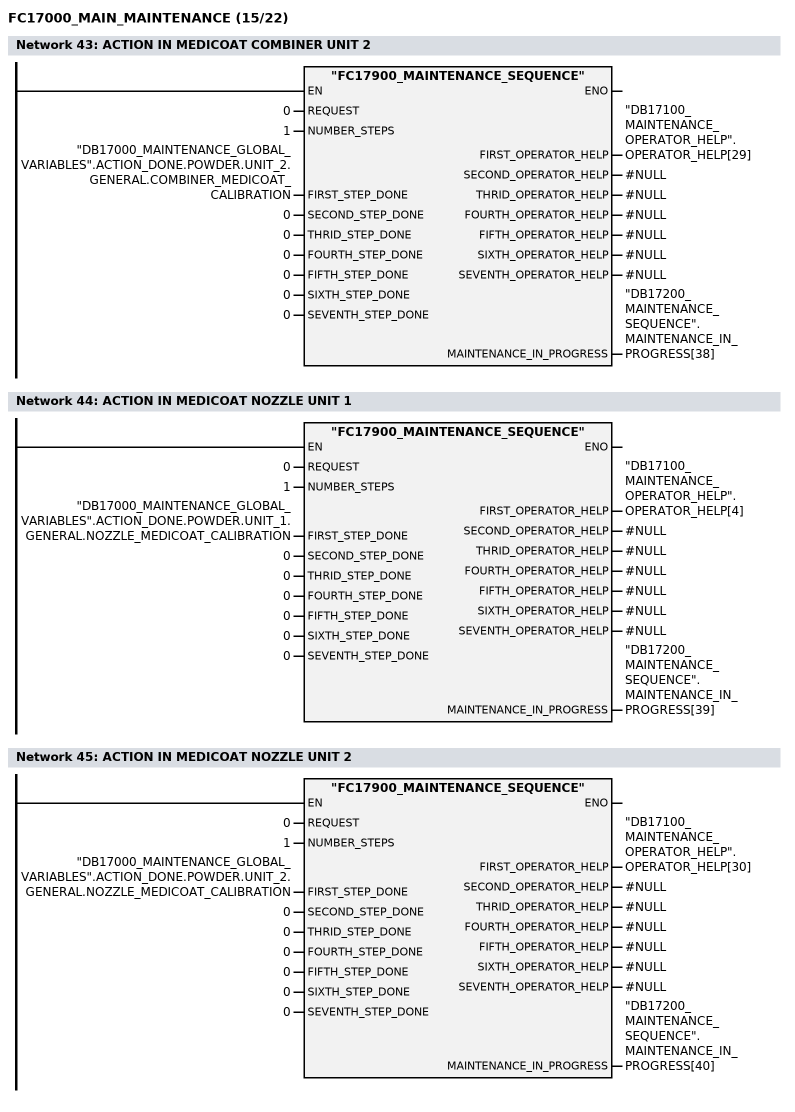
   RUNG wire#powerrail
      "FC17900_MAINTENANCE_SEQUENCE"(REQUEST := 0, NUMBER_STEPS := 1, FIRST_STEP_DONE := "DB17000_MAINTENANCE_GLOBAL_VARIABLES".ACTION_DONE.POWDER.UNIT_2.GENERAL.COMBINER_MEDICOAT_CALIBRATION, SECOND_STEP_DONE := 0, THRID_STEP_DONE := 0, FOURTH_STEP_DONE := 0, FIFTH_STEP_DONE := 0, SIXTH_STEP_DONE := 0, SEVENTH_STEP_DONE := 0, FIRST_OPERATOR_HELP => "DB17100_MAINTENANCE_OPERATOR_HELP".OPERATOR_HELP[29], SECOND_OPERATOR_HELP => #NULL, THRID_OPERATOR_HELP => #NULL, FOURTH_OPERATOR_HELP => #NULL, FIFTH_OPERATOR_HELP => #NULL, SIXTH_OPERATOR_HELP => #NULL, SEVENTH_OPERATOR_HELP => #NULL, MAINTENANCE_IN_PROGRESS => "DB17200_MAINTENANCE_SEQUENCE".MAINTENANCE_IN_PROGRESS[38])
   END_RUNG
   // the same network as SCL:
   "FC17900_MAINTENANCE_SEQUENCE"(REQUEST := 0,
                           NUMBER_STEPS := 1,
                           FIRST_STEP_DONE := "DB17000_MAINTENANCE_GLOBAL_VARIABLES".ACTION_DONE.POWDER.UNIT_2.GENERAL.COMBINER_MEDICOAT_CALIBRATION,
                           SECOND_STEP_DONE := 0,
                           THRID_STEP_DONE := 0,
                           FOURTH_STEP_DONE := 0,
                           FIFTH_STEP_DONE := 0,
                           SIXTH_STEP_DONE := 0,
                           SEVENTH_STEP_DONE := 0,
                           FIRST_OPERATOR_HELP => "DB17100_MAINTENANCE_OPERATOR_HELP".OPERATOR_HELP[29],
                           SECOND_OPERATOR_HELP => #NULL,
                           THRID_OPERATOR_HELP => #NULL,
                           FOURTH_OPERATOR_HELP => #NULL,
                           FIFTH_OPERATOR_HELP => #NULL,
                           SIXTH_OPERATOR_HELP => #NULL,
                           SEVENTH_OPERATOR_HELP => #NULL,
                           MAINTENANCE_IN_PROGRESS => "DB17200_MAINTENANCE_SEQUENCE".MAINTENANCE_IN_PROGRESS[38]);
END_REGION

REGION Network 44: ACTION IN MEDICOAT NOZZLE UNIT 1
   RUNG wire#powerrail
      "FC17900_MAINTENANCE_SEQUENCE"(REQUEST := 0, NUMBER_STEPS := 1, FIRST_STEP_DONE := "DB17000_MAINTENANCE_GLOBAL_VARIABLES".ACTION_DONE.POWDER.UNIT_1.GENERAL.NOZZLE_MEDICOAT_CALIBRATION, SECOND_STEP_DONE := 0, THRID_STEP_DONE := 0, FOURTH_STEP_DONE := 0, FIFTH_STEP_DONE := 0, SIXTH_STEP_DONE := 0, SEVENTH_STEP_DONE := 0, FIRST_OPERATOR_HELP => "DB17100_MAINTENANCE_OPERATOR_HELP".OPERATOR_HELP[4], SECOND_OPERATOR_HELP => #NULL, THRID_OPERATOR_HELP => #NULL, FOURTH_OPERATOR_HELP => #NULL, FIFTH_OPERATOR_HELP => #NULL, SIXTH_OPERATOR_HELP => #NULL, SEVENTH_OPERATOR_HELP => #NULL, MAINTENANCE_IN_PROGRESS => "DB17200_MAINTENANCE_SEQUENCE".MAINTENANCE_IN_PROGRESS[39])
   END_RUNG
   // the same network as SCL:
   "FC17900_MAINTENANCE_SEQUENCE"(REQUEST := 0,
                           NUMBER_STEPS := 1,
                           FIRST_STEP_DONE := "DB17000_MAINTENANCE_GLOBAL_VARIABLES".ACTION_DONE.POWDER.UNIT_1.GENERAL.NOZZLE_MEDICOAT_CALIBRATION,
                           SECOND_STEP_DONE := 0,
                           THRID_STEP_DONE := 0,
                           FOURTH_STEP_DONE := 0,
                           FIFTH_STEP_DONE := 0,
                           SIXTH_STEP_DONE := 0,
                           SEVENTH_STEP_DONE := 0,
                           FIRST_OPERATOR_HELP => "DB17100_MAINTENANCE_OPERATOR_HELP".OPERATOR_HELP[4],
                           SECOND_OPERATOR_HELP => #NULL,
                           THRID_OPERATOR_HELP => #NULL,
                           FOURTH_OPERATOR_HELP => #NULL,
                           FIFTH_OPERATOR_HELP => #NULL,
                           SIXTH_OPERATOR_HELP => #NULL,
                           SEVENTH_OPERATOR_HELP => #NULL,
                           MAINTENANCE_IN_PROGRESS => "DB17200_MAINTENANCE_SEQUENCE".MAINTENANCE_IN_PROGRESS[39]);
END_REGION

REGION Network 45: ACTION IN MEDICOAT NOZZLE UNIT 2
   RUNG wire#powerrail
      "FC17900_MAINTENANCE_SEQUENCE"(REQUEST := 0, NUMBER_STEPS := 1, FIRST_STEP_DONE := "DB17000_MAINTENANCE_GLOBAL_VARIABLES".ACTION_DONE.POWDER.UNIT_2.GENERAL.NOZZLE_MEDICOAT_CALIBRATION, SECOND_STEP_DONE := 0, THRID_STEP_DONE := 0, FOURTH_STEP_DONE := 0, FIFTH_STEP_DONE := 0, SIXTH_STEP_DONE := 0, SEVENTH_STEP_DONE := 0, FIRST_OPERATOR_HELP => "DB17100_MAINTENANCE_OPERATOR_HELP".OPERATOR_HELP[30], SECOND_OPERATOR_HELP => #NULL, THRID_OPERATOR_HELP => #NULL, FOURTH_OPERATOR_HELP => #NULL, FIFTH_OPERATOR_HELP => #NULL, SIXTH_OPERATOR_HELP => #NULL, SEVENTH_OPERATOR_HELP => #NULL, MAINTENANCE_IN_PROGRESS => "DB17200_MAINTENANCE_SEQUENCE".MAINTENANCE_IN_PROGRESS[40])
   END_RUNG
   // the same network as SCL:
   "FC17900_MAINTENANCE_SEQUENCE"(REQUEST := 0,
                           NUMBER_STEPS := 1,
                           FIRST_STEP_DONE := "DB17000_MAINTENANCE_GLOBAL_VARIABLES".ACTION_DONE.POWDER.UNIT_2.GENERAL.NOZZLE_MEDICOAT_CALIBRATION,
                           SECOND_STEP_DONE := 0,
                           THRID_STEP_DONE := 0,
                           FOURTH_STEP_DONE := 0,
                           FIFTH_STEP_DONE := 0,
                           SIXTH_STEP_DONE := 0,
                           SEVENTH_STEP_DONE := 0,
                           FIRST_OPERATOR_HELP => "DB17100_MAINTENANCE_OPERATOR_HELP".OPERATOR_HELP[30],
                           SECOND_OPERATOR_HELP => #NULL,
                           THRID_OPERATOR_HELP => #NULL,
                           FOURTH_OPERATOR_HELP => #NULL,
                           FIFTH_OPERATOR_HELP => #NULL,
                           SIXTH_OPERATOR_HELP => #NULL,
                           SEVENTH_OPERATOR_HELP => #NULL,
                           MAINTENANCE_IN_PROGRESS => "DB17200_MAINTENANCE_SEQUENCE".MAINTENANCE_IN_PROGRESS[40]);
END_REGION

REGION Network 46: ACTION IN LOADING CELL UNIT 1
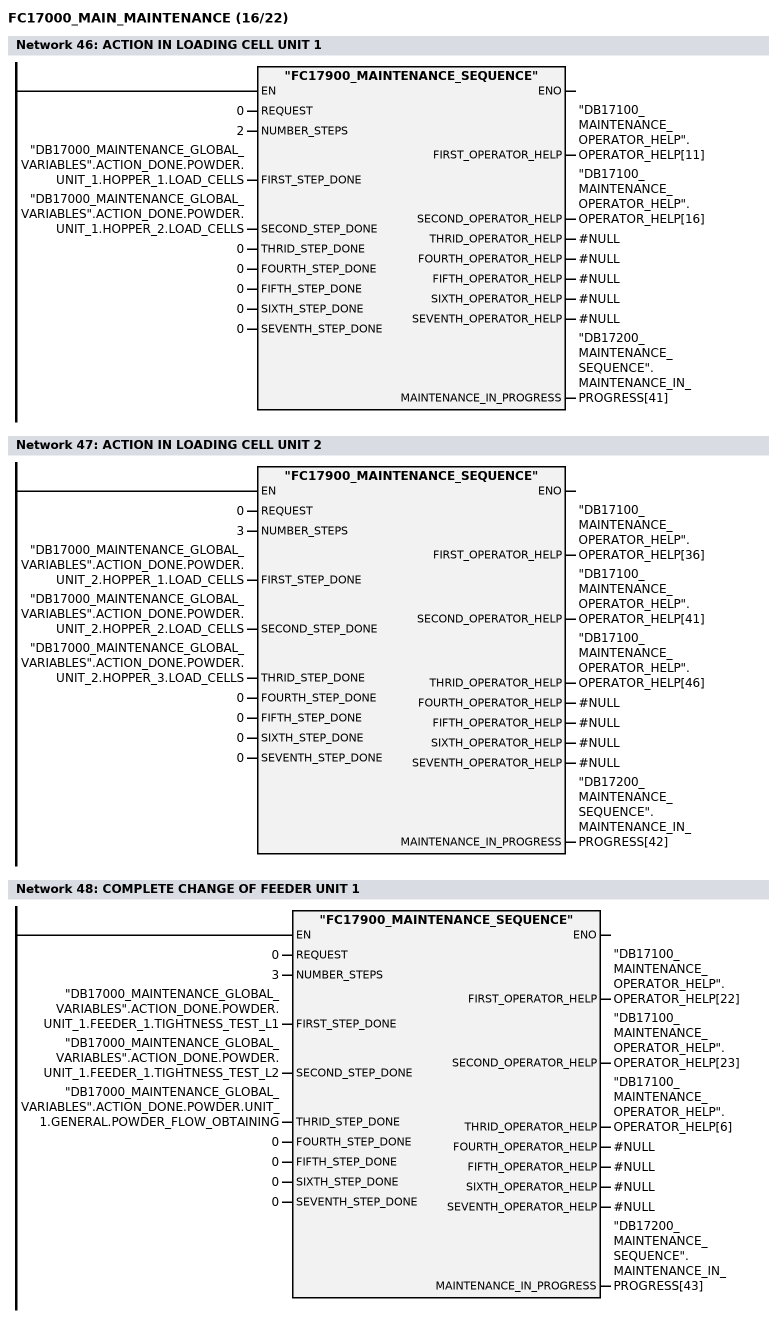
   RUNG wire#powerrail
      "FC17900_MAINTENANCE_SEQUENCE"(REQUEST := 0, NUMBER_STEPS := 2, FIRST_STEP_DONE := "DB17000_MAINTENANCE_GLOBAL_VARIABLES".ACTION_DONE.POWDER.UNIT_1.HOPPER_1.LOAD_CELLS, SECOND_STEP_DONE := "DB17000_MAINTENANCE_GLOBAL_VARIABLES".ACTION_DONE.POWDER.UNIT_1.HOPPER_2.LOAD_CELLS, THRID_STEP_DONE := 0, FOURTH_STEP_DONE := 0, FIFTH_STEP_DONE := 0, SIXTH_STEP_DONE := 0, SEVENTH_STEP_DONE := 0, FIRST_OPERATOR_HELP => "DB17100_MAINTENANCE_OPERATOR_HELP".OPERATOR_HELP[11], SECOND_OPERATOR_HELP => "DB17100_MAINTENANCE_OPERATOR_HELP".OPERATOR_HELP[16], THRID_OPERATOR_HELP => #NULL, FOURTH_OPERATOR_HELP => #NULL, FIFTH_OPERATOR_HELP => #NULL, SIXTH_OPERATOR_HELP => #NULL, SEVENTH_OPERATOR_HELP => #NULL, MAINTENANCE_IN_PROGRESS => "DB17200_MAINTENANCE_SEQUENCE".MAINTENANCE_IN_PROGRESS[41])
   END_RUNG
   // the same network as SCL:
   "FC17900_MAINTENANCE_SEQUENCE"(REQUEST := 0,
                           NUMBER_STEPS := 2,
                           FIRST_STEP_DONE := "DB17000_MAINTENANCE_GLOBAL_VARIABLES".ACTION_DONE.POWDER.UNIT_1.HOPPER_1.LOAD_CELLS,
                           SECOND_STEP_DONE := "DB17000_MAINTENANCE_GLOBAL_VARIABLES".ACTION_DONE.POWDER.UNIT_1.HOPPER_2.LOAD_CELLS,
                           THRID_STEP_DONE := 0,
                           FOURTH_STEP_DONE := 0,
                           FIFTH_STEP_DONE := 0,
                           SIXTH_STEP_DONE := 0,
                           SEVENTH_STEP_DONE := 0,
                           FIRST_OPERATOR_HELP => "DB17100_MAINTENANCE_OPERATOR_HELP".OPERATOR_HELP[11],
                           SECOND_OPERATOR_HELP => "DB17100_MAINTENANCE_OPERATOR_HELP".OPERATOR_HELP[16],
                           THRID_OPERATOR_HELP => #NULL,
                           FOURTH_OPERATOR_HELP => #NULL,
                           FIFTH_OPERATOR_HELP => #NULL,
                           SIXTH_OPERATOR_HELP => #NULL,
                           SEVENTH_OPERATOR_HELP => #NULL,
                           MAINTENANCE_IN_PROGRESS => "DB17200_MAINTENANCE_SEQUENCE".MAINTENANCE_IN_PROGRESS[41]);
END_REGION

